FUNCTION_BLOCK "fbVFD_GSeries"   // FB120, LAD
TITLE = Controls a Siemens G120 VFD (or MicroMaster)
{ S7_Optimized_Access := 'TRUE' }
VERSION : 0.1
// stored: AutoNumber false, IsIECCheckEnabled false, IsRetainMemResEnabled false, MemoryReserve 100, SetENOAutomatically false, UDAEnableTagReadback false
   VAR_INPUT
      tInTimeout { ExternalAccessible := 'False'; ExternalVisible := 'False'; ExternalWritable := 'False'} : Time;   // Timeout Time
      iInMode { ExternalAccessible := 'False'; ExternalVisible := 'False'; ExternalWritable := 'False'} : Int;   // Mode Selection
      hwInTelegram { ExternalAccessible := 'False'; ExternalVisible := 'False'; ExternalWritable := 'False'} : HW_SUBMODULE;   // VFD Standard Telegram 1 HW address
      bInEstop { ExternalAccessible := 'False'; ExternalVisible := 'False'; ExternalWritable := 'False'} : Bool;   // Estop
      bInSignalContactor { ExternalAccessible := 'False'; ExternalVisible := 'False'; ExternalWritable := 'False'} : Bool;   // Feedback signal from Contactor
      bInEnableForward { ExternalAccessible := 'False'; ExternalVisible := 'False'; ExternalWritable := 'False'} : Bool;   // Forward motion enebled
      bInEnableReverse { ExternalAccessible := 'False'; ExternalVisible := 'False'; ExternalWritable := 'False'} : Bool := false;   // Reverse motion enabled
      rInCommandSpeed { ExternalAccessible := 'False'; ExternalVisible := 'False'; ExternalWritable := 'False'} : Real;   // Auto mode speed SP
      bInCommandForward { ExternalAccessible := 'False'; ExternalVisible := 'False'; ExternalWritable := 'False'} : Bool;   // Move forward in automatic mode
      bInCommandReverse { ExternalAccessible := 'False'; ExternalVisible := 'False'; ExternalWritable := 'False'} : Bool := false;   // Move Reverse in automatic mode
      bInResetError { ExternalAccessible := 'False'; ExternalVisible := 'False'; ExternalWritable := 'False'} : Bool;   // Reset Error
      bInMotorProtector { ExternalAccessible := 'False'; ExternalVisible := 'False'; ExternalWritable := 'False'} : Bool := true;   // Motor Protector input
      bInLocalDisconnect { ExternalAccessible := 'False'; ExternalVisible := 'False'; ExternalWritable := 'False'} : Bool := true;   // Local switch input
      bInClutch { ExternalAccessible := 'False'; ExternalVisible := 'False'; ExternalWritable := 'False'} : Bool := true;   // Overload clutch
      bInCoolingFan { ExternalAccessible := 'False'; ExternalVisible := 'False'; ExternalWritable := 'False'} : Bool := true;   // Cooling fan input
      bInUseCurrentAlarm { ExternalAccessible := 'False'; ExternalVisible := 'False'; ExternalWritable := 'False'} : Bool := false;   // True if current alarm should be active
      bInUseMaxFrequencyAlarm { ExternalAccessible := 'False'; ExternalVisible := 'False'; ExternalWritable := 'False'} : Bool := false;   // True is max frequency alarm should be active
      bInSimulate { ExternalAccessible := 'False'; ExternalVisible := 'False'; ExternalWritable := 'False'} : Bool := false;   // Activate device simulation
   END_VAR
   VAR_OUTPUT
      rOutSpeed { ExternalAccessible := 'False'; ExternalVisible := 'False'; ExternalWritable := 'False'} : Real;   // Actual motor speed
      bOutContactor { ExternalAccessible := 'False'; ExternalVisible := 'False'; ExternalWritable := 'False'} : Bool;   // Motor contactor ON
      bOutCommandForward { ExternalAccessible := 'False'; ExternalVisible := 'False'; ExternalWritable := 'False'} : Bool;   // Motor forward command
      bOutCommandReverse { ExternalAccessible := 'False'; ExternalVisible := 'False'; ExternalWritable := 'False'} : Bool := false;   // Motor reverse command
      bOutActiveForward { ExternalAccessible := 'False'; ExternalVisible := 'False'; ExternalWritable := 'False'} : Bool;   // Motor is running forward
      bOutActiveReverse { ExternalAccessible := 'False'; ExternalVisible := 'False'; ExternalWritable := 'False'} : Bool;   // Motor is running backward
      bOutAuto { ExternalAccessible := 'False'; ExternalVisible := 'False'; ExternalWritable := 'False'} : Bool;   // Block in auto mode
      bOutError { ExternalAccessible := 'False'; ExternalVisible := 'False'; ExternalWritable := 'False'} : Bool;   // Error exists
      ERROR_VFD { ExternalAccessible := 'False'; ExternalVisible := 'False'; ExternalWritable := 'False'} : "udtError_VFD";   // UDT Structure for VFD errors
   END_VAR
   VAR_IN_OUT
      HMI_VFD_Control : "udtHMI_VFD_Control";   // UDT Structure for VFD HMI control
   END_VAR
   VAR
      ErrorScroller { ExternalAccessible := 'False'; ExternalVisible := 'False'; ExternalWritable := 'False'; S7_SetPoint := 'True'} : "fbErrorScroller";   // fb to control scrolling of errors on HMI
      TON_TimeOut { ExternalAccessible := 'False'; ExternalVisible := 'False'; ExternalWritable := 'False'; S7_SetPoint := 'True'} : TON_TIME;   // Timer for Timeout time
      TON_ContactorDelay { ExternalAccessible := 'False'; ExternalVisible := 'False'; ExternalWritable := 'False'; S7_SetPoint := 'True'} : TON_TIME;   // Contactor on delay timer before check errors
      TON_CoolingFan { ExternalAccessible := 'False'; ExternalVisible := 'False'; ExternalWritable := 'False'; S7_SetPoint := 'True'} : TON_TIME;
      TON_CurrentLimitDebounce { ExternalAccessible := 'False'; ExternalVisible := 'False'; ExternalWritable := 'False'; S7_SetPoint := 'True'} : TON_TIME;   // Debounce timer for current at limit
      iLastMode { ExternalAccessible := 'False'; ExternalVisible := 'False'; ExternalWritable := 'False'} : Int;   // Last mode code
      wStatusWord { ExternalAccessible := 'False'; ExternalVisible := 'False'; ExternalWritable := 'False'} : Word;   // VFD Status word
      iActualSpeed { ExternalAccessible := 'False'; ExternalVisible := 'False'; ExternalWritable := 'False'} : Int;   // VFD Actual speed
      wControlWord { ExternalAccessible := 'False'; ExternalVisible := 'False'; ExternalWritable := 'False'} : Word;   // VFD Control word output
      iSpeedSetPoint { ExternalAccessible := 'False'; ExternalVisible := 'False'; ExternalWritable := 'False'} : Int;   // VFD Speed output
      rCommandSpeed { ExternalAccessible := 'False'; ExternalVisible := 'False'; ExternalWritable := 'False'} : Real;   // Speed command
      bNewMode { ExternalAccessible := 'False'; ExternalVisible := 'False'; ExternalWritable := 'False'} : Bool;   // New mode selected
      bEnableForward { ExternalAccessible := 'False'; ExternalVisible := 'False'; ExternalWritable := 'False'} : Bool;   // Forward enabled
      bEnableReverse { ExternalAccessible := 'False'; ExternalVisible := 'False'; ExternalWritable := 'False'} : Bool;   // Reverse enabled
      bManualMode { ExternalAccessible := 'False'; ExternalVisible := 'False'; ExternalWritable := 'False'} : Bool;   // Manual Mode is Active
      bAutoMode { ExternalAccessible := 'False'; ExternalVisible := 'False'; ExternalWritable := 'False'} : Bool;   // Auto Mode is Active
      bRunTimeoutTimer { ExternalAccessible := 'False'; ExternalVisible := 'False'; ExternalWritable := 'False'} : Bool;   // run the timeout timer
      bReset { ExternalAccessible := 'False'; ExternalVisible := 'False'; ExternalWritable := 'False'} : Bool;
      bTON_TimeOut { ExternalAccessible := 'False'; ExternalVisible := 'False'; ExternalWritable := 'False'} : Bool;
      bTON_ContactorDelay { ExternalAccessible := 'False'; ExternalVisible := 'False'; ExternalWritable := 'False'} : Bool;
      bTON_CoolingFan { ExternalAccessible := 'False'; ExternalVisible := 'False'; ExternalWritable := 'False'} : Bool;
      bTON_CurrentLimitDebounce { ExternalAccessible := 'False'; ExternalVisible := 'False'; ExternalWritable := 'False'} : Bool;
      bPB_Forward { ExternalAccessible := 'False'; ExternalVisible := 'False'; ExternalWritable := 'False'} : Bool;
      bPB_Reverse { ExternalAccessible := 'False'; ExternalVisible := 'False'; ExternalWritable := 'False'} : Bool;
      bPB_Stop { ExternalAccessible := 'False'; ExternalVisible := 'False'; ExternalWritable := 'False'} : Bool;
      bPB_ResetError { ExternalAccessible := 'False'; ExternalVisible := 'False'; ExternalWritable := 'False'} : Bool;
   END_VAR
   VAR_TEMP
      CONTROL : Struct   // VFD Control Structure
         bON : Bool;   // On
         bOFF2 : Bool;   // Off2
         bOFF3 : Bool;   // Off3
         bENABLE_OPERATION : Bool;   // Enable Operation
         bDISABLE_RFG : Bool;   // Disable RFG
         bENABLE_RFG : Bool;   // Enable RFG
         bSETPOINT_ENABLE : Bool;   // Setpoint Enable
         bFAULT_ACK : Bool;   // Fault Acknowledge
         bCW_ACTIVATION : Bool;   // CW Activation
         bCCW_ACTIVATION : Bool;   // CCW Activation
         bSP_VALID : Bool;   // SP Valid
         bSP_INVERTED : Bool;   // SP Inverted
         bSPARE01 : Bool;   // Spare
         bMOTOR_POT_UP : Bool;   // Motor Pot up
         bMOTOR_POT_DN : Bool;   // Motor Pot down
         bLOCAL_ACTIVE : Bool;   // Local Active
      END_STRUCT;
      STATUS : Struct   // VFD Status Structure
         bAT_SETPOINT_FREQ : Bool;   // At Setpoint Frequency
         bMASTER_CONTROL : Bool;   // Master Control
         bMAX_FREQ_REACHED : Bool;   // Max Frequency Reached
         bCURRENT_LIMIT : Bool;   // Current Limit
         bBRAKE_ACTIVE : Bool;   // Brake Active
         bMOTOR_OVERLOAD : Bool;   // Motor Overload
         bCW_ROTATION : Bool;   // CW Rotation
         bINVERTER_OVERLOAD : Bool;   // Inverter Overload
         bREADY_FOR_ENABLE : Bool;   // Ready for Enable
         bREADY_TO_RUN : Bool;   // Ready To Run
         bRUNNING : Bool;   // Running
         bFAULT : Bool;   // Fault
         bOFF2_ACTIVE : Bool;   // Off2 Active
         bOFF3_ACTIVE : Bool;   // Off3 Active
         bSTART_LOCKOUT : Bool;   // Start Lockout
         bALARM : Bool;   // Alarm
      END_STRUCT;
      bMajorFault : Bool;   // Major Fault
      arrReadTemp : Array[1..6] of Word;
      dwWriteTemp : DWord;   // temporary dword
      bTemp : Bool;   // temp bit
      wTempWordValue : Word;   // used for temporaily holding a word value
      iTemp : Word;
      rTemp : Real;   // temporary real value
      tTemp : Time;   // temp time value
   END_VAR
   VAR CONSTANT
      crMaxSetPoint : Real := 200.0;   // Maximum speed set point
      crMinSetPoint : Real := 0.0;   // Minimum speed set point
      crSpeedScaling : Real := 163.84;   // Reference speed scale value
   END_VAR
   VAR_TEMP   // added for the SCL form of the ladder/FBD networks
      _w1 : Bool;
      _w2 : Bool;
      _w3 : Bool;
      _w4 : Bool;
   END_VAR
BEGIN

REGION Network 1: --------------------------------------------------------- Inputs ------------------------------------------------------------------
END_REGION

REGION Network 2: Read HMI input buttons
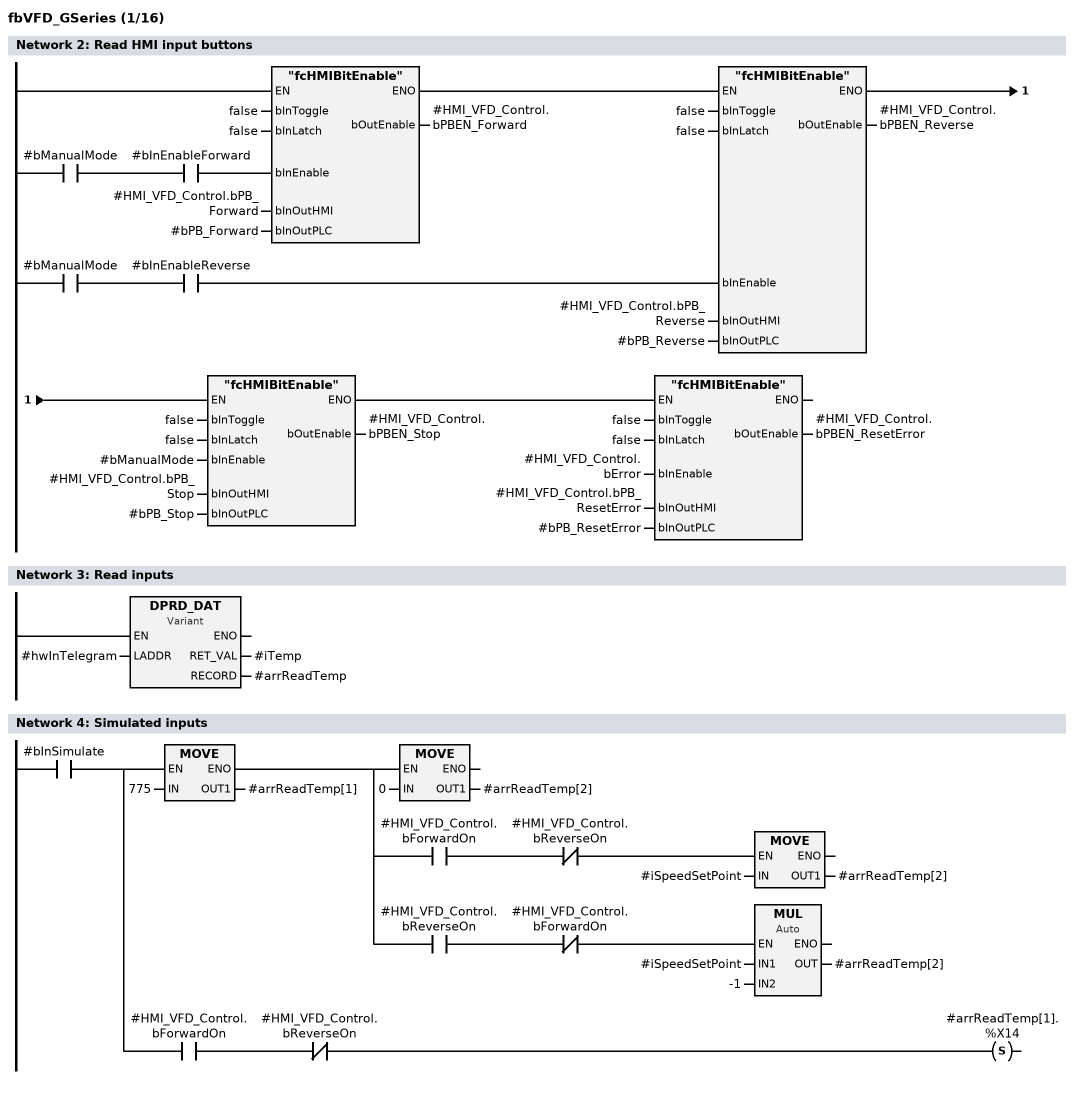
   RUNG wire#powerrail
      "fcHMIBitEnable"(bInEnable := wire#w1, bInToggle := false, bInLatch := false, bInOutHMI := #HMI_VFD_Control.bPB_Forward, bInOutPLC := #bPB_Forward, bOutEnable => #HMI_VFD_Control.bPBEN_Forward)
      "fcHMIBitEnable"(bInEnable := wire#w2, bInToggle := false, bInLatch := false, bInOutHMI := #HMI_VFD_Control.bPB_Reverse, bInOutPLC := #bPB_Reverse, bOutEnable => #HMI_VFD_Control.bPBEN_Reverse)
      "fcHMIBitEnable"(bInToggle := false, bInLatch := false, bInEnable := #bManualMode, bInOutHMI := #HMI_VFD_Control.bPB_Stop, bInOutPLC := #bPB_Stop, bOutEnable => #HMI_VFD_Control.bPBEN_Stop)
      "fcHMIBitEnable"(bInToggle := false, bInLatch := false, bInEnable := #HMI_VFD_Control.bError, bInOutHMI := #HMI_VFD_Control.bPB_ResetError, bInOutPLC := #bPB_ResetError, bOutEnable => #HMI_VFD_Control.bPBEN_ResetError)
   END_RUNG
   RUNG wire#powerrail
      Contact( #bManualMode )
      Contact( #bInEnableForward )
   END_RUNG wire#w1
   RUNG wire#powerrail
      Contact( #bManualMode )
      Contact( #bInEnableReverse )
   END_RUNG wire#w2
   // the same network as SCL:
   "fcHMIBitEnable"(bInToggle := false,
                    bInLatch := false,
                    bInEnable := #bManualMode AND #bInEnableForward,
                    bInOutHMI := #HMI_VFD_Control.bPB_Forward,
                    bInOutPLC := #bPB_Forward,
                    bOutEnable => #HMI_VFD_Control.bPBEN_Forward,
                    ENO => #_w1);
   "fcHMIBitEnable"(EN := #_w1,
                    bInToggle := false,
                    bInLatch := false,
                    bInEnable := #bManualMode AND #bInEnableReverse,
                    bInOutHMI := #HMI_VFD_Control.bPB_Reverse,
                    bInOutPLC := #bPB_Reverse,
                    bOutEnable => #HMI_VFD_Control.bPBEN_Reverse,
                    ENO => #_w2);
   "fcHMIBitEnable"(EN := #_w2,
                    bInToggle := false,
                    bInLatch := false,
                    bInEnable := #bManualMode,
                    bInOutHMI := #HMI_VFD_Control.bPB_Stop,
                    bInOutPLC := #bPB_Stop,
                    bOutEnable => #HMI_VFD_Control.bPBEN_Stop,
                    ENO => #_w3);
   IF #_w3 THEN
       "fcHMIBitEnable"(bInToggle := false,
                        bInLatch := false,
                        bInEnable := #HMI_VFD_Control.bError,
                        bInOutHMI := #HMI_VFD_Control.bPB_ResetError,
                        bInOutPLC := #bPB_ResetError,
                        bOutEnable => #HMI_VFD_Control.bPBEN_ResetError);
   END_IF;
END_REGION

REGION Network 3: Read inputs
   RUNG wire#powerrail
      { S7_Templates := "[ptr_type := Variant, laddr_type := HW_IO]" } DPRD_DAT(LADDR := #hwInTelegram, RET_VAL => #iTemp, RECORD => #arrReadTemp)
   END_RUNG
   // the same network as SCL:
   #iTemp := DPRD_DAT(LADDR := #hwInTelegram, RECORD => #arrReadTemp);
END_REGION

REGION Network 4: Simulated inputs
   RUNG wire#powerrail
      Contact( #bInSimulate )
      wire#w1
      Move(in := 775, out1 => #arrReadTemp[1])
      wire#w2
      Move(in := 0, out1 => #arrReadTemp[2])
   END_RUNG
   RUNG wire#w2
      Contact( #HMI_VFD_Control.bForwardOn )
      I_Contact( #HMI_VFD_Control.bReverseOn )
      Move(in := #iSpeedSetPoint, out1 => #arrReadTemp[2])
   END_RUNG
   RUNG wire#w2
      Contact( #HMI_VFD_Control.bReverseOn )
      I_Contact( #HMI_VFD_Control.bForwardOn )
      Mul(in1 := #iSpeedSetPoint, in2 := -1, out => #arrReadTemp[2])
   END_RUNG
   RUNG wire#w1
      Contact( #HMI_VFD_Control.bForwardOn )
      I_Contact( #HMI_VFD_Control.bReverseOn )
      S_Coil( #arrReadTemp[1].%X14 )
   END_RUNG
   // the same network as SCL:
   IF #bInSimulate THEN
       #arrReadTemp[1] := 775;
       #arrReadTemp[2] := 0;
   END_IF;
   IF #bInSimulate AND #HMI_VFD_Control.bForwardOn AND NOT #HMI_VFD_Control.bReverseOn THEN
       #arrReadTemp[2] := #iSpeedSetPoint;
   END_IF;
   IF #bInSimulate AND #HMI_VFD_Control.bReverseOn AND NOT #HMI_VFD_Control.bForwardOn THEN
       #arrReadTemp[2] := #iSpeedSetPoint * (-1);
   END_IF;
   IF #bInSimulate AND #HMI_VFD_Control.bForwardOn AND NOT #HMI_VFD_Control.bReverseOn THEN
       #arrReadTemp[1].%X14 := TRUE;
   END_IF;
END_REGION

REGION Network 5: Read the status word and parse to bits
   // // Read status word.  First word at iInAddress is the status word
   // wStatusWord := PIW[iInAddress];
   // 
   // fcWordToBits( wIN_WORD                    := wStatusWord,  // Parse status word
   //                 bOUT_BIT00                  := STATUS.bREADY_FOR_ENABLE,
   //                 bOUT_BIT01                  := STATUS.bREADY_TO_RUN,
   //                 bOUT_BIT02                  := STATUS.bRUNNING,
   //                 bOUT_BIT03                  := STATUS.bFAULT,
   //                 bOUT_BIT04                  := STATUS.bOFF2_ACTIVE,
   //                 bOUT_BIT05                  := STATUS.bOFF3_ACTIVE,
   //                 bOUT_BIT06                  := STATUS.bSTART_LOCKOUT,
   //                 bOUT_BIT07                  := STATUS.bALARM,
   //                 bOUT_BIT08                  := STATUS.bAT_SETPOINT_FREQ,
   //                 bOUT_BIT09                  := STATUS.bMASTER_CONTROL,
   //                 bOUT_BIT10                  := STATUS.bMAX_FREQ_REACHED,
   //                 bOUT_BIT11                  := STATUS.bCURRENT_LIMIT,
   //                 bOUT_BIT12                  := STATUS.bBRAKE_ACTIVE,
   //                 bOUT_BIT13                  := STATUS.bMOTOR_OVERLOAD,
   //                 bOUT_BIT14                  := STATUS.bCW_ROTATION,
   //                 bOUT_BIT15                  := STATUS.bINVERTER_OVERLOAD);
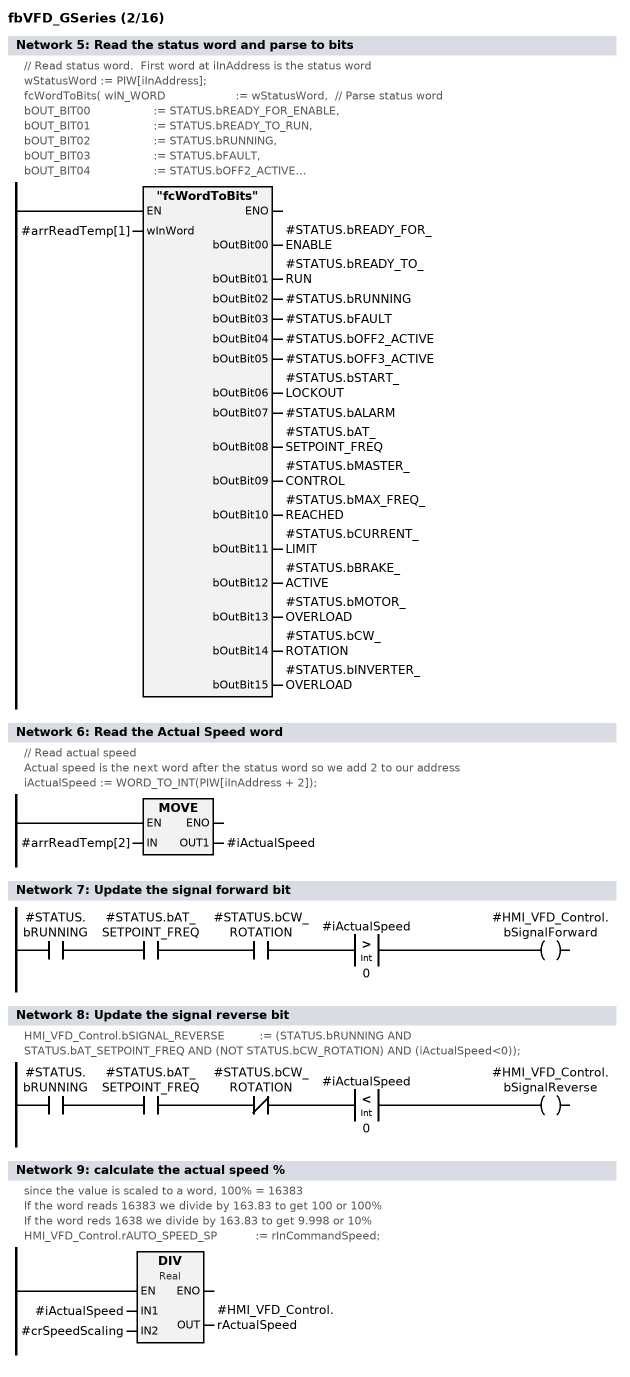
   RUNG wire#powerrail
      "fcWordToBits"(wInWord := #arrReadTemp[1], bOutBit00 => #STATUS.bREADY_FOR_ENABLE, bOutBit01 => #STATUS.bREADY_TO_RUN, bOutBit02 => #STATUS.bRUNNING, bOutBit03 => #STATUS.bFAULT, bOutBit04 => #STATUS.bOFF2_ACTIVE, bOutBit05 => #STATUS.bOFF3_ACTIVE, bOutBit06 => #STATUS.bSTART_LOCKOUT, bOutBit07 => #STATUS.bALARM, bOutBit08 => #STATUS.bAT_SETPOINT_FREQ, bOutBit09 => #STATUS.bMASTER_CONTROL, bOutBit10 => #STATUS.bMAX_FREQ_REACHED, bOutBit11 => #STATUS.bCURRENT_LIMIT, bOutBit12 => #STATUS.bBRAKE_ACTIVE, bOutBit13 => #STATUS.bMOTOR_OVERLOAD, bOutBit14 => #STATUS.bCW_ROTATION, bOutBit15 => #STATUS.bINVERTER_OVERLOAD)
   END_RUNG
   // the same network as SCL:
   "fcWordToBits"(wInWord := #arrReadTemp[1],
                  bOutBit00 => #STATUS.bREADY_FOR_ENABLE,
                  bOutBit01 => #STATUS.bREADY_TO_RUN,
                  bOutBit02 => #STATUS.bRUNNING,
                  bOutBit03 => #STATUS.bFAULT,
                  bOutBit04 => #STATUS.bOFF2_ACTIVE,
                  bOutBit05 => #STATUS.bOFF3_ACTIVE,
                  bOutBit06 => #STATUS.bSTART_LOCKOUT,
                  bOutBit07 => #STATUS.bALARM,
                  bOutBit08 => #STATUS.bAT_SETPOINT_FREQ,
                  bOutBit09 => #STATUS.bMASTER_CONTROL,
                  bOutBit10 => #STATUS.bMAX_FREQ_REACHED,
                  bOutBit11 => #STATUS.bCURRENT_LIMIT,
                  bOutBit12 => #STATUS.bBRAKE_ACTIVE,
                  bOutBit13 => #STATUS.bMOTOR_OVERLOAD,
                  bOutBit14 => #STATUS.bCW_ROTATION,
                  bOutBit15 => #STATUS.bINVERTER_OVERLOAD);
END_REGION

REGION Network 6: Read the Actual Speed word
   // // Read actual speed
   // Actual speed is the next word after the status word so we add 2 to our address
   // iActualSpeed := WORD_TO_INT(PIW[iInAddress + 2]);
   RUNG wire#powerrail
      Move(in := #arrReadTemp[2], out1 => #iActualSpeed)
   END_RUNG
   // the same network as SCL:
   #iActualSpeed := #arrReadTemp[2];
END_REGION

REGION Network 7: Update the signal forward bit
   RUNG wire#powerrail
      Contact( #STATUS.bRUNNING )
      Contact( #STATUS.bAT_SETPOINT_FREQ )
      Contact( #STATUS.bCW_ROTATION )
      { S7_Templates := "SrcType := Int" } GT_Contact(in1 := #iActualSpeed, in2 := 0)
      Coil( #HMI_VFD_Control.bSignalForward )
   END_RUNG
   // the same network as SCL:
   #HMI_VFD_Control.bSignalForward := #STATUS.bRUNNING AND #STATUS.bAT_SETPOINT_FREQ AND #STATUS.bCW_ROTATION AND (#iActualSpeed > 0);
END_REGION

REGION Network 8: Update the signal reverse bit
   // HMI_VFD_Control.bSIGNAL_REVERSE          := (STATUS.bRUNNING AND 
   // STATUS.bAT_SETPOINT_FREQ AND (NOT STATUS.bCW_ROTATION) AND (iActualSpeed<0));
   RUNG wire#powerrail
      Contact( #STATUS.bRUNNING )
      Contact( #STATUS.bAT_SETPOINT_FREQ )
      I_Contact( #STATUS.bCW_ROTATION )
      { S7_Templates := "SrcType := Int" } LT_Contact(in1 := #iActualSpeed, in2 := 0)
      Coil( #HMI_VFD_Control.bSignalReverse )
   END_RUNG
   // the same network as SCL:
   #HMI_VFD_Control.bSignalReverse := #STATUS.bRUNNING AND #STATUS.bAT_SETPOINT_FREQ AND NOT #STATUS.bCW_ROTATION AND (#iActualSpeed < 0);
END_REGION

REGION Network 9: calculate the actual speed %
   // since the value is scaled to a word, 100% = 16383
   // 
   // If the word reads 16383 we divide by 163.83 to get 100 or 100%
   // If the word reds 1638 we divide by 163.83 to get 9.998 or 10%
   // 
   // HMI_VFD_Control.rAUTO_SPEED_SP           := rInCommandSpeed;
   RUNG wire#powerrail
      { S7_Templates := "SrcType := Real" } Div(in1 := #iActualSpeed, in2 := #crSpeedScaling, out => #HMI_VFD_Control.rActualSpeed)
   END_RUNG
   // the same network as SCL:
   #HMI_VFD_Control.rActualSpeed := #iActualSpeed / #crSpeedScaling;
END_REGION

REGION Network 10: Set the automatic mode speed set point
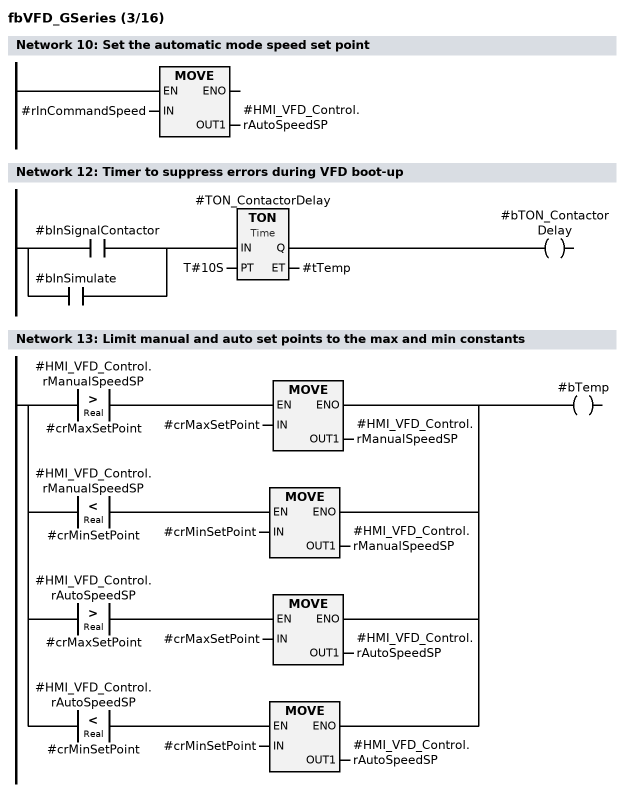
   RUNG wire#powerrail
      Move(in := #rInCommandSpeed, out1 => #HMI_VFD_Control.rAutoSpeedSP)
   END_RUNG
   // the same network as SCL:
   #HMI_VFD_Control.rAutoSpeedSP := #rInCommandSpeed;
END_REGION

REGION Network 11: --------------------------------------------------- Control Logic ------------------------------------------------------------
END_REGION

REGION Network 12: Timer to suppress errors during VFD boot-up
   RUNG wire#powerrail
      Contact( #bInSignalContactor )
      wire#w1
      { S7_Templates := "time_type := Time" } #TON_ContactorDelay.TON(pt := T#10S, et => #tTemp)
      Coil( #bTON_ContactorDelay )
   END_RUNG
   RUNG wire#powerrail
      Contact( #bInSimulate )
   END_RUNG wire#w1
   // the same network as SCL:
   #TON_ContactorDelay(IN := #bInSignalContactor OR #bInSimulate, PT := T#10S, ET => #tTemp);   // TON
   #bTON_ContactorDelay := #TON_ContactorDelay.Q;
END_REGION

REGION Network 13: Limit manual and auto set points to the max and min constants
   RUNG wire#powerrail
      { S7_Templates := "SrcType := Real" } GT_Contact(in1 := #HMI_VFD_Control.rManualSpeedSP, in2 := #crMaxSetPoint)
      Move(in := #crMaxSetPoint, out1 => #HMI_VFD_Control.rManualSpeedSP)
      wire#w1
      Coil( #bTemp )
   END_RUNG
   RUNG wire#powerrail
      { S7_Templates := "SrcType := Real" } LT_Contact(in1 := #HMI_VFD_Control.rManualSpeedSP, in2 := #crMinSetPoint)
      Move(in := #crMinSetPoint, out1 => #HMI_VFD_Control.rManualSpeedSP)
   END_RUNG wire#w1
   RUNG wire#powerrail
      { S7_Templates := "SrcType := Real" } GT_Contact(in1 := #HMI_VFD_Control.rAutoSpeedSP, in2 := #crMaxSetPoint)
      Move(in := #crMaxSetPoint, out1 => #HMI_VFD_Control.rAutoSpeedSP)
   END_RUNG wire#w1
   RUNG wire#powerrail
      { S7_Templates := "SrcType := Real" } LT_Contact(in1 := #HMI_VFD_Control.rAutoSpeedSP, in2 := #crMinSetPoint)
      Move(in := #crMinSetPoint, out1 => #HMI_VFD_Control.rAutoSpeedSP)
   END_RUNG wire#w1
   // the same network as SCL:
   #_w1 := #HMI_VFD_Control.rManualSpeedSP > #crMaxSetPoint;
   IF #_w1 THEN #HMI_VFD_Control.rManualSpeedSP := #crMaxSetPoint; END_IF;
   #_w2 := #HMI_VFD_Control.rManualSpeedSP < #crMinSetPoint;
   IF #_w2 THEN #HMI_VFD_Control.rManualSpeedSP := #crMinSetPoint; END_IF;
   #_w3 := #HMI_VFD_Control.rAutoSpeedSP > #crMaxSetPoint;
   IF #_w3 THEN #HMI_VFD_Control.rAutoSpeedSP := #crMaxSetPoint; END_IF;
   #_w4 := #HMI_VFD_Control.rAutoSpeedSP < #crMinSetPoint;
   IF #_w4 THEN #HMI_VFD_Control.rAutoSpeedSP := #crMinSetPoint; END_IF;
   #bTemp := #_w1 OR #_w2 OR #_w3 OR #_w4;
END_REGION

REGION Network 14: Reset errors
   // Clear all errors
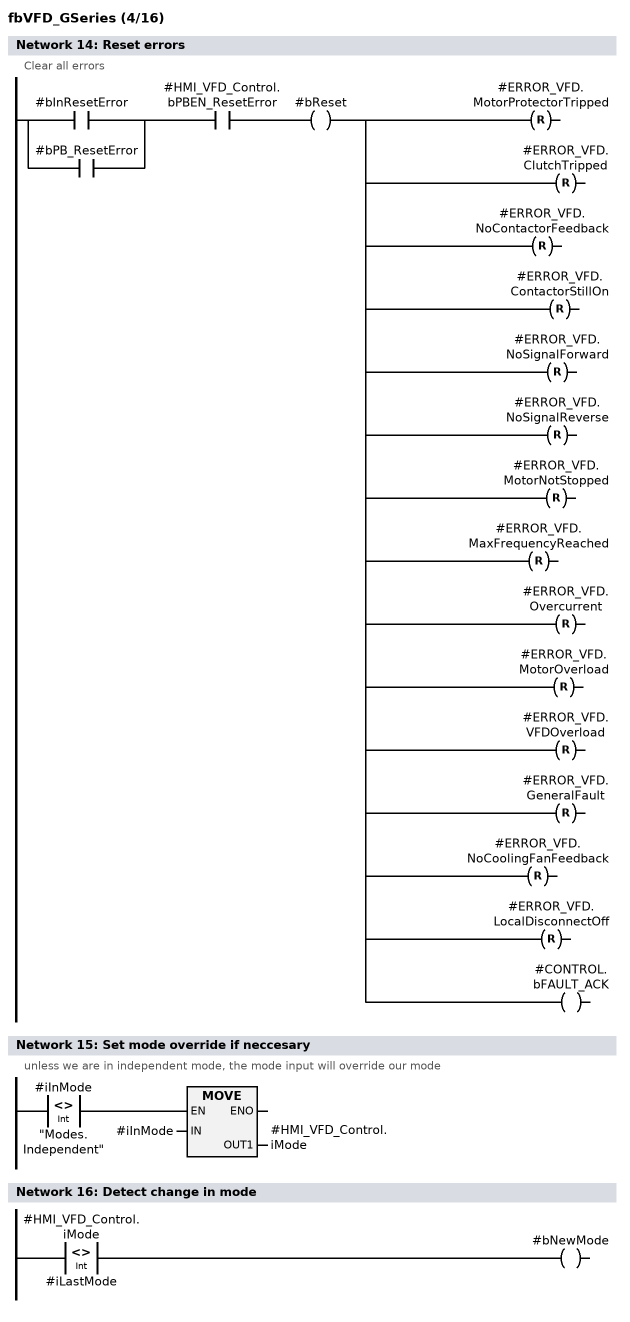
   RUNG wire#powerrail
      Contact( #bInResetError )
      wire#w1
      Contact( #HMI_VFD_Control.bPBEN_ResetError )
      Coil( #bReset )
      wire#w2
      R_Coil( #ERROR_VFD.MotorProtectorTripped )
   END_RUNG
   RUNG wire#powerrail
      Contact( #bPB_ResetError )
   END_RUNG wire#w1
   RUNG wire#w2
      R_Coil( #ERROR_VFD.ClutchTripped )
   END_RUNG
   RUNG wire#w2
      R_Coil( #ERROR_VFD.NoContactorFeedback )
   END_RUNG
   RUNG wire#w2
      R_Coil( #ERROR_VFD.ContactorStillOn )
   END_RUNG
   RUNG wire#w2
      R_Coil( #ERROR_VFD.NoSignalForward )
   END_RUNG
   RUNG wire#w2
      R_Coil( #ERROR_VFD.NoSignalReverse )
   END_RUNG
   RUNG wire#w2
      R_Coil( #ERROR_VFD.MotorNotStopped )
   END_RUNG
   RUNG wire#w2
      R_Coil( #ERROR_VFD.MaxFrequencyReached )
   END_RUNG
   RUNG wire#w2
      R_Coil( #ERROR_VFD.Overcurrent )
   END_RUNG
   RUNG wire#w2
      R_Coil( #ERROR_VFD.MotorOverload )
   END_RUNG
   RUNG wire#w2
      R_Coil( #ERROR_VFD.VFDOverload )
   END_RUNG
   RUNG wire#w2
      R_Coil( #ERROR_VFD.GeneralFault )
   END_RUNG
   RUNG wire#w2
      R_Coil( #ERROR_VFD.NoCoolingFanFeedback )
   END_RUNG
   RUNG wire#w2
      R_Coil( #ERROR_VFD.LocalDisconnectOff )
   END_RUNG
   RUNG wire#w2
      Coil( #CONTROL.bFAULT_ACK )
   END_RUNG
   // the same network as SCL:
   #bReset := (#bInResetError OR #bPB_ResetError) AND #HMI_VFD_Control.bPBEN_ResetError;
   IF #bReset THEN
       #ERROR_VFD.MotorProtectorTripped := FALSE;
       #ERROR_VFD.ClutchTripped := FALSE;
       #ERROR_VFD.NoContactorFeedback := FALSE;
       #ERROR_VFD.ContactorStillOn := FALSE;
       #ERROR_VFD.NoSignalForward := FALSE;
       #ERROR_VFD.NoSignalReverse := FALSE;
       #ERROR_VFD.MotorNotStopped := FALSE;
       #ERROR_VFD.MaxFrequencyReached := FALSE;
       #ERROR_VFD.Overcurrent := FALSE;
       #ERROR_VFD.MotorOverload := FALSE;
       #ERROR_VFD.VFDOverload := FALSE;
       #ERROR_VFD.GeneralFault := FALSE;
       #ERROR_VFD.NoCoolingFanFeedback := FALSE;
       #ERROR_VFD.LocalDisconnectOff := FALSE;
   END_IF;
   #CONTROL.bFAULT_ACK := #bReset;
END_REGION

REGION Network 15: Set mode override if neccesary
   // unless we are in independent mode, the mode input will override our mode
   RUNG wire#powerrail
      { S7_Templates := "SrcType := Int" } NE_Contact(in1 := #iInMode, in2 := "Modes.Independent")
      Move(in := #iInMode, out1 => #HMI_VFD_Control.iMode)
   END_RUNG
   // the same network as SCL:
   IF #iInMode <> "Modes.Independent" THEN #HMI_VFD_Control.iMode := #iInMode; END_IF;
END_REGION

REGION Network 16: Detect change in mode
   RUNG wire#powerrail
      { S7_Templates := "SrcType := Int" } NE_Contact(in1 := #HMI_VFD_Control.iMode, in2 := #iLastMode)
      Coil( #bNewMode )
   END_RUNG
   // the same network as SCL:
   #bNewMode := #HMI_VFD_Control.iMode <> #iLastMode;
END_REGION

REGION Network 17: Keep track of last mode
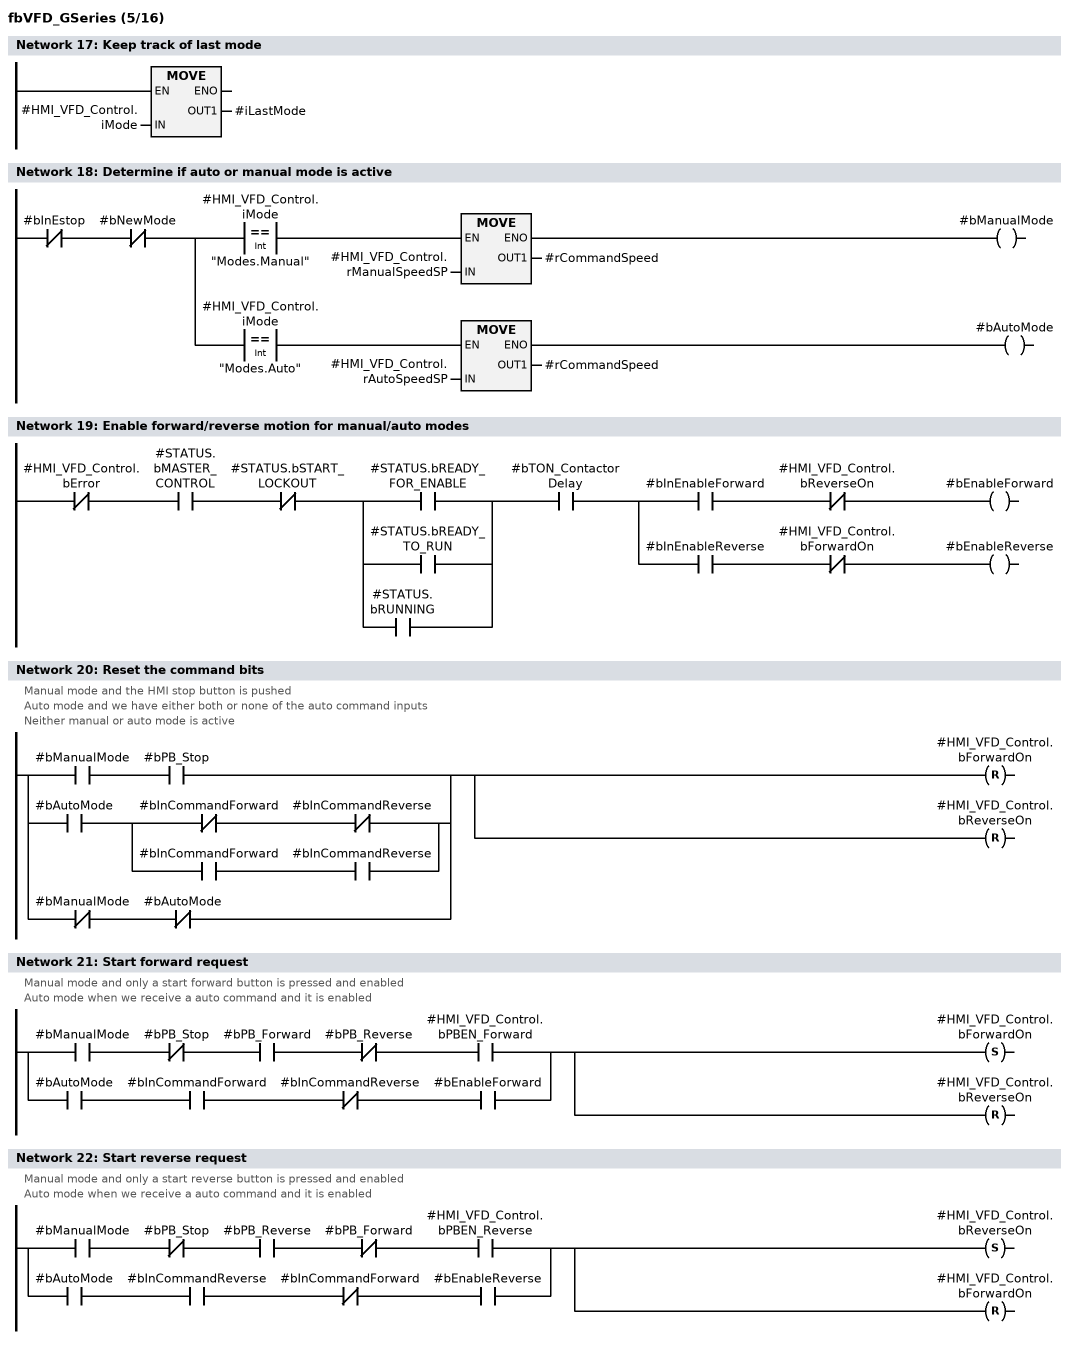
   RUNG wire#powerrail
      Move(in := #HMI_VFD_Control.iMode, out1 => #iLastMode)
   END_RUNG
   // the same network as SCL:
   #iLastMode := #HMI_VFD_Control.iMode;
END_REGION

REGION Network 18: Determine if auto or manual mode is active
   RUNG wire#powerrail
      I_Contact( #bInEstop )
      I_Contact( #bNewMode )
      wire#w1
      { S7_Templates := "SrcType := Int" } EQ_Contact(in1 := #HMI_VFD_Control.iMode, in2 := "Modes.Manual")
      Move(in := #HMI_VFD_Control.rManualSpeedSP, out1 => #rCommandSpeed)
      Coil( #bManualMode )
   END_RUNG
   RUNG wire#w1
      { S7_Templates := "SrcType := Int" } EQ_Contact(in1 := #HMI_VFD_Control.iMode, in2 := "Modes.Auto")
      Move(in := #HMI_VFD_Control.rAutoSpeedSP, out1 => #rCommandSpeed)
      Coil( #bAutoMode )
   END_RUNG
   // the same network as SCL:
   #_w1 := NOT #bInEstop AND NOT #bNewMode;
   #_w2 := #_w1 AND (#HMI_VFD_Control.iMode = "Modes.Manual");
   IF #_w2 THEN #rCommandSpeed := #HMI_VFD_Control.rManualSpeedSP; END_IF;
   #bManualMode := #_w2;
   #_w3 := #_w1 AND (#HMI_VFD_Control.iMode = "Modes.Auto");
   IF #_w3 THEN #rCommandSpeed := #HMI_VFD_Control.rAutoSpeedSP; END_IF;
   #bAutoMode := #_w3;
END_REGION

REGION Network 19: Enable forward/reverse motion for manual/auto modes
   RUNG wire#powerrail
      I_Contact( #HMI_VFD_Control.bError )
      Contact( #STATUS.bMASTER_CONTROL )
      I_Contact( #STATUS.bSTART_LOCKOUT )
      wire#w1
      Contact( #STATUS.bREADY_FOR_ENABLE )
      wire#w2
      Contact( #bTON_ContactorDelay )
      wire#w3
      Contact( #bInEnableForward )
      I_Contact( #HMI_VFD_Control.bReverseOn )
      Coil( #bEnableForward )
   END_RUNG
   RUNG wire#w1
      Contact( #STATUS.bREADY_TO_RUN )
   END_RUNG wire#w2
   RUNG wire#w1
      Contact( #STATUS.bRUNNING )
   END_RUNG wire#w2
   RUNG wire#w3
      Contact( #bInEnableReverse )
      I_Contact( #HMI_VFD_Control.bForwardOn )
      Coil( #bEnableReverse )
   END_RUNG
   // the same network as SCL:
   #_w1 := NOT #HMI_VFD_Control.bError AND #STATUS.bMASTER_CONTROL AND NOT #STATUS.bSTART_LOCKOUT AND (#STATUS.bREADY_FOR_ENABLE OR #STATUS.bREADY_TO_RUN OR #STATUS.bRUNNING) AND #bTON_ContactorDelay;
   #bEnableForward := #_w1 AND #bInEnableForward AND NOT #HMI_VFD_Control.bReverseOn;
   #bEnableReverse := #_w1 AND #bInEnableReverse AND NOT #HMI_VFD_Control.bForwardOn;
END_REGION

REGION Network 20: Reset the command bits
   // Manual mode and the HMI stop button is pushed
   // Auto mode and we have either both or none of the auto command inputs
   // Neither manual or auto mode is active
   RUNG wire#powerrail
      Contact( #bManualMode )
      Contact( #bPB_Stop )
      wire#w1
      R_Coil( #HMI_VFD_Control.bForwardOn )
   END_RUNG
   RUNG wire#powerrail
      Contact( #bAutoMode )
      wire#w2
      I_Contact( #bInCommandForward )
      I_Contact( #bInCommandReverse )
   END_RUNG wire#w1
   RUNG wire#w2
      Contact( #bInCommandForward )
      Contact( #bInCommandReverse )
   END_RUNG wire#w1
   RUNG wire#powerrail
      I_Contact( #bManualMode )
      I_Contact( #bAutoMode )
   END_RUNG wire#w1
   RUNG wire#w1
      R_Coil( #HMI_VFD_Control.bReverseOn )
   END_RUNG
   // the same network as SCL:
   IF (#bManualMode AND #bPB_Stop) OR (#bAutoMode AND ((NOT #bInCommandForward AND NOT #bInCommandReverse) OR (#bInCommandForward AND #bInCommandReverse))) OR (NOT #bManualMode AND NOT #bAutoMode) THEN
       #HMI_VFD_Control.bForwardOn := FALSE;
       #HMI_VFD_Control.bReverseOn := FALSE;
   END_IF;
END_REGION

REGION Network 21: Start forward request
   // Manual mode and only a start forward button is pressed and enabled
   // Auto mode when we receive a auto command and it is enabled
   RUNG wire#powerrail
      Contact( #bManualMode )
      I_Contact( #bPB_Stop )
      Contact( #bPB_Forward )
      I_Contact( #bPB_Reverse )
      Contact( #HMI_VFD_Control.bPBEN_Forward )
      wire#w1
      S_Coil( #HMI_VFD_Control.bForwardOn )
   END_RUNG
   RUNG wire#powerrail
      Contact( #bAutoMode )
      Contact( #bInCommandForward )
      I_Contact( #bInCommandReverse )
      Contact( #bEnableForward )
   END_RUNG wire#w1
   RUNG wire#w1
      R_Coil( #HMI_VFD_Control.bReverseOn )
   END_RUNG
   // the same network as SCL:
   IF (#bManualMode AND NOT #bPB_Stop AND #bPB_Forward AND NOT #bPB_Reverse AND #HMI_VFD_Control.bPBEN_Forward) OR (#bAutoMode AND #bInCommandForward AND NOT #bInCommandReverse AND #bEnableForward) THEN
       #HMI_VFD_Control.bForwardOn := TRUE;
       #HMI_VFD_Control.bReverseOn := FALSE;
   END_IF;
END_REGION

REGION Network 22: Start reverse request
   // Manual mode and only a start reverse button is pressed and enabled
   // Auto mode when we receive a auto command and it is enabled
   RUNG wire#powerrail
      Contact( #bManualMode )
      I_Contact( #bPB_Stop )
      Contact( #bPB_Reverse )
      I_Contact( #bPB_Forward )
      Contact( #HMI_VFD_Control.bPBEN_Reverse )
      wire#w1
      S_Coil( #HMI_VFD_Control.bReverseOn )
   END_RUNG
   RUNG wire#powerrail
      Contact( #bAutoMode )
      Contact( #bInCommandReverse )
      I_Contact( #bInCommandForward )
      Contact( #bEnableReverse )
   END_RUNG wire#w1
   RUNG wire#w1
      R_Coil( #HMI_VFD_Control.bForwardOn )
   END_RUNG
   // the same network as SCL:
   IF (#bManualMode AND NOT #bPB_Stop AND #bPB_Reverse AND NOT #bPB_Forward AND #HMI_VFD_Control.bPBEN_Reverse) OR (#bAutoMode AND #bInCommandReverse AND NOT #bInCommandForward AND #bEnableReverse) THEN
       #HMI_VFD_Control.bReverseOn := TRUE;
       #HMI_VFD_Control.bForwardOn := FALSE;
   END_IF;
END_REGION

REGION Network 23: If the forward enable is lost, stop the forward motion
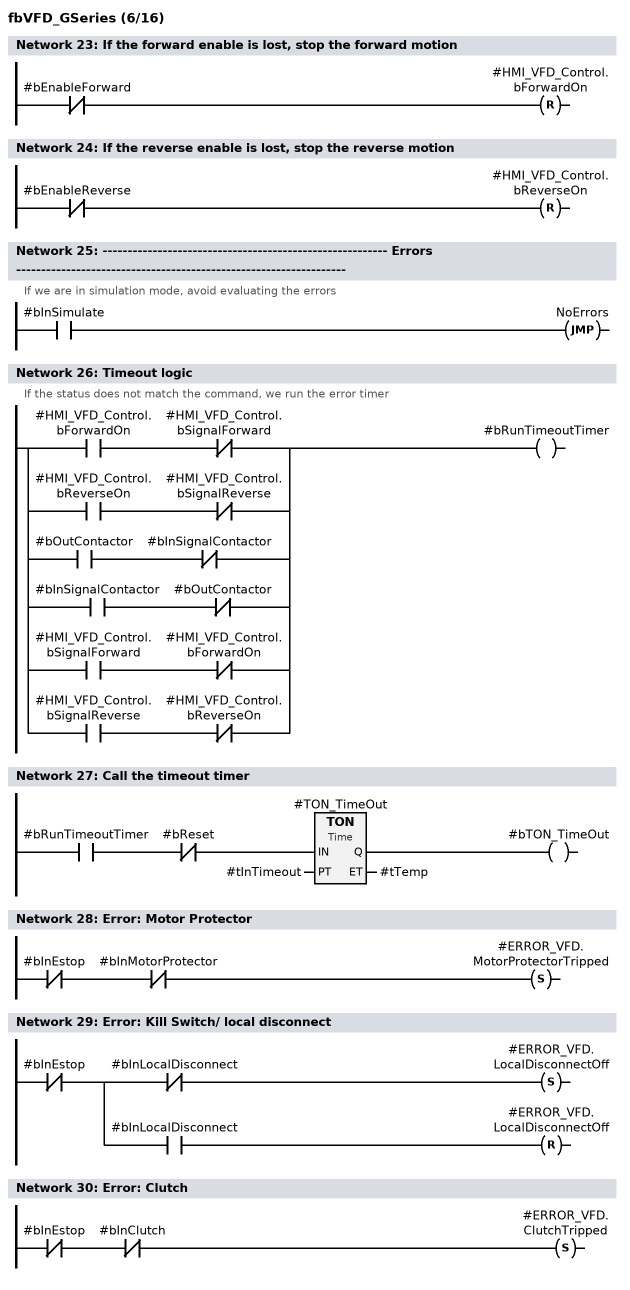
   RUNG wire#powerrail
      I_Contact( #bEnableForward )
      R_Coil( #HMI_VFD_Control.bForwardOn )
   END_RUNG
   // the same network as SCL:
   IF NOT #bEnableForward THEN #HMI_VFD_Control.bForwardOn := FALSE; END_IF;
END_REGION

REGION Network 24: If the reverse enable is lost, stop the reverse motion
   RUNG wire#powerrail
      I_Contact( #bEnableReverse )
      R_Coil( #HMI_VFD_Control.bReverseOn )
   END_RUNG
   // the same network as SCL:
   IF NOT #bEnableReverse THEN #HMI_VFD_Control.bReverseOn := FALSE; END_IF;
END_REGION

REGION Network 25: --------------------------------------------------------- Errors ------------------------------------------------------------------
   // If we are in simulation mode, avoid evaluating the errors
   RUNG wire#powerrail
      Contact( #bInSimulate )
      JumpCoil( NoErrors )
   END_RUNG
   // the same network as SCL:
   IF #bInSimulate THEN GOTO NoErrors; END_IF;
END_REGION

REGION Network 26: Timeout logic
   // If the status does not match the command, we run the error timer
   RUNG wire#powerrail
      Contact( #HMI_VFD_Control.bForwardOn )
      I_Contact( #HMI_VFD_Control.bSignalForward )
      wire#w1
      Coil( #bRunTimeoutTimer )
   END_RUNG
   RUNG wire#powerrail
      Contact( #HMI_VFD_Control.bReverseOn )
      I_Contact( #HMI_VFD_Control.bSignalReverse )
   END_RUNG wire#w1
   RUNG wire#powerrail
      Contact( #bOutContactor )
      I_Contact( #bInSignalContactor )
   END_RUNG wire#w1
   RUNG wire#powerrail
      Contact( #bInSignalContactor )
      I_Contact( #bOutContactor )
   END_RUNG wire#w1
   RUNG wire#powerrail
      Contact( #HMI_VFD_Control.bSignalForward )
      I_Contact( #HMI_VFD_Control.bForwardOn )
   END_RUNG wire#w1
   RUNG wire#powerrail
      Contact( #HMI_VFD_Control.bSignalReverse )
      I_Contact( #HMI_VFD_Control.bReverseOn )
   END_RUNG wire#w1
   // the same network as SCL:
   #bRunTimeoutTimer := (#HMI_VFD_Control.bForwardOn AND NOT #HMI_VFD_Control.bSignalForward) OR (#HMI_VFD_Control.bReverseOn AND NOT #HMI_VFD_Control.bSignalReverse) OR (#bOutContactor AND NOT #bInSignalContactor) OR (#bInSignalContactor AND NOT #bOutContactor) OR (#HMI_VFD_Control.bSignalForward AND NOT #HMI_VFD_Control.bForwardOn) OR (#HMI_VFD_Control.bSignalReverse AND NOT #HMI_VFD_Control.bReverseOn);
END_REGION

REGION Network 27: Call the timeout timer
   RUNG wire#powerrail
      Contact( #bRunTimeoutTimer )
      I_Contact( #bReset )
      { S7_Templates := "time_type := Time" } #TON_TimeOut.TON(pt := #tInTimeout, et => #tTemp)
      Coil( #bTON_TimeOut )
   END_RUNG
   // the same network as SCL:
   #TON_TimeOut(IN := #bRunTimeoutTimer AND NOT #bReset, PT := #tInTimeout, ET => #tTemp);   // TON
   #bTON_TimeOut := #TON_TimeOut.Q;
END_REGION

REGION Network 28: Error: Motor Protector
   RUNG wire#powerrail
      I_Contact( #bInEstop )
      I_Contact( #bInMotorProtector )
      S_Coil( #ERROR_VFD.MotorProtectorTripped )
   END_RUNG
   // the same network as SCL:
   IF NOT #bInEstop AND NOT #bInMotorProtector THEN #ERROR_VFD.MotorProtectorTripped := TRUE; END_IF;
END_REGION

REGION Network 29: Error: Kill Switch/ local disconnect
   RUNG wire#powerrail
      I_Contact( #bInEstop )
      wire#w1
      I_Contact( #bInLocalDisconnect )
      S_Coil( #ERROR_VFD.LocalDisconnectOff )
   END_RUNG
   RUNG wire#w1
      Contact( #bInLocalDisconnect )
      R_Coil( #ERROR_VFD.LocalDisconnectOff )
   END_RUNG
   // the same network as SCL:
   IF NOT #bInEstop AND NOT #bInLocalDisconnect THEN #ERROR_VFD.LocalDisconnectOff := TRUE; END_IF;
   IF NOT #bInEstop AND #bInLocalDisconnect THEN #ERROR_VFD.LocalDisconnectOff := FALSE; END_IF;
END_REGION

REGION Network 30: Error: Clutch
   RUNG wire#powerrail
      I_Contact( #bInEstop )
      I_Contact( #bInClutch )
      S_Coil( #ERROR_VFD.ClutchTripped )
   END_RUNG
   // the same network as SCL:
   IF NOT #bInEstop AND NOT #bInClutch THEN #ERROR_VFD.ClutchTripped := TRUE; END_IF;
END_REGION

REGION Network 31: Error: Max Frequency. This error isn't always used.
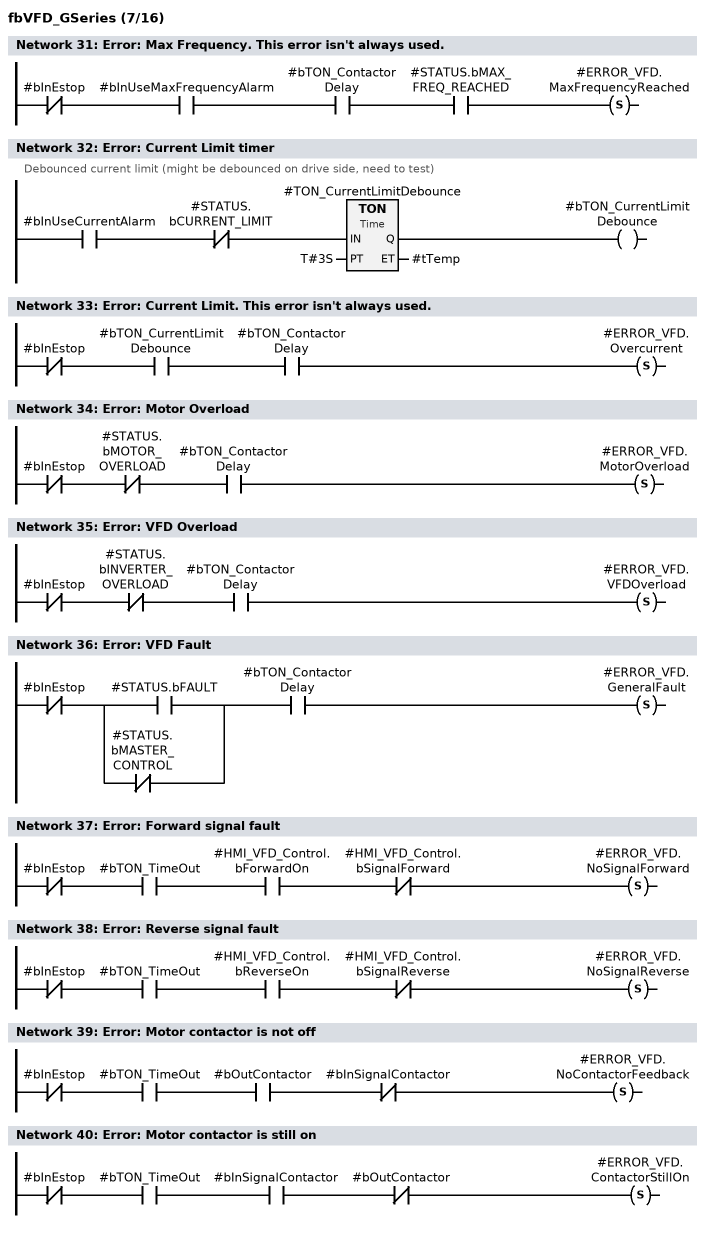
   RUNG wire#powerrail
      I_Contact( #bInEstop )
      Contact( #bInUseMaxFrequencyAlarm )
      Contact( #bTON_ContactorDelay )
      Contact( #STATUS.bMAX_FREQ_REACHED )
      S_Coil( #ERROR_VFD.MaxFrequencyReached )
   END_RUNG
   // the same network as SCL:
   IF NOT #bInEstop AND #bInUseMaxFrequencyAlarm AND #bTON_ContactorDelay AND #STATUS.bMAX_FREQ_REACHED THEN
       #ERROR_VFD.MaxFrequencyReached := TRUE;
   END_IF;
END_REGION

REGION Network 32: Error: Current Limit timer
   // Debounced current limit (might be debounced on drive side, need to test)
   RUNG wire#powerrail
      Contact( #bInUseCurrentAlarm )
      I_Contact( #STATUS.bCURRENT_LIMIT )
      { S7_Templates := "time_type := Time" } #TON_CurrentLimitDebounce.TON(pt := T#3S, et => #tTemp)
      Coil( #bTON_CurrentLimitDebounce )
   END_RUNG
   // the same network as SCL:
   #TON_CurrentLimitDebounce(IN := #bInUseCurrentAlarm AND NOT #STATUS.bCURRENT_LIMIT, PT := T#3S, ET => #tTemp);   // TON
   #bTON_CurrentLimitDebounce := #TON_CurrentLimitDebounce.Q;
END_REGION

REGION Network 33: Error: Current Limit. This error isn't always used.
   RUNG wire#powerrail
      I_Contact( #bInEstop )
      Contact( #bTON_CurrentLimitDebounce )
      Contact( #bTON_ContactorDelay )
      S_Coil( #ERROR_VFD.Overcurrent )
   END_RUNG
   // the same network as SCL:
   IF NOT #bInEstop AND #bTON_CurrentLimitDebounce AND #bTON_ContactorDelay THEN
       #ERROR_VFD.Overcurrent := TRUE;
   END_IF;
END_REGION

REGION Network 34: Error: Motor Overload
   RUNG wire#powerrail
      I_Contact( #bInEstop )
      I_Contact( #STATUS.bMOTOR_OVERLOAD )
      Contact( #bTON_ContactorDelay )
      S_Coil( #ERROR_VFD.MotorOverload )
   END_RUNG
   // the same network as SCL:
   IF NOT #bInEstop AND NOT #STATUS.bMOTOR_OVERLOAD AND #bTON_ContactorDelay THEN
       #ERROR_VFD.MotorOverload := TRUE;
   END_IF;
END_REGION

REGION Network 35: Error: VFD Overload
   RUNG wire#powerrail
      I_Contact( #bInEstop )
      I_Contact( #STATUS.bINVERTER_OVERLOAD )
      Contact( #bTON_ContactorDelay )
      S_Coil( #ERROR_VFD.VFDOverload )
   END_RUNG
   // the same network as SCL:
   IF NOT #bInEstop AND NOT #STATUS.bINVERTER_OVERLOAD AND #bTON_ContactorDelay THEN
       #ERROR_VFD.VFDOverload := TRUE;
   END_IF;
END_REGION

REGION Network 36: Error: VFD Fault
   RUNG wire#powerrail
      I_Contact( #bInEstop )
      wire#w1
      Contact( #STATUS.bFAULT )
      wire#w2
      Contact( #bTON_ContactorDelay )
      S_Coil( #ERROR_VFD.GeneralFault )
   END_RUNG
   RUNG wire#w1
      I_Contact( #STATUS.bMASTER_CONTROL )
   END_RUNG wire#w2
   // the same network as SCL:
   IF NOT #bInEstop AND (#STATUS.bFAULT OR NOT #STATUS.bMASTER_CONTROL) AND #bTON_ContactorDelay THEN
       #ERROR_VFD.GeneralFault := TRUE;
   END_IF;
END_REGION

REGION Network 37: Error: Forward signal fault
   RUNG wire#powerrail
      I_Contact( #bInEstop )
      Contact( #bTON_TimeOut )
      Contact( #HMI_VFD_Control.bForwardOn )
      I_Contact( #HMI_VFD_Control.bSignalForward )
      S_Coil( #ERROR_VFD.NoSignalForward )
   END_RUNG
   // the same network as SCL:
   IF NOT #bInEstop AND #bTON_TimeOut AND #HMI_VFD_Control.bForwardOn AND NOT #HMI_VFD_Control.bSignalForward THEN
       #ERROR_VFD.NoSignalForward := TRUE;
   END_IF;
END_REGION

REGION Network 38: Error: Reverse signal fault
   RUNG wire#powerrail
      I_Contact( #bInEstop )
      Contact( #bTON_TimeOut )
      Contact( #HMI_VFD_Control.bReverseOn )
      I_Contact( #HMI_VFD_Control.bSignalReverse )
      S_Coil( #ERROR_VFD.NoSignalReverse )
   END_RUNG
   // the same network as SCL:
   IF NOT #bInEstop AND #bTON_TimeOut AND #HMI_VFD_Control.bReverseOn AND NOT #HMI_VFD_Control.bSignalReverse THEN
       #ERROR_VFD.NoSignalReverse := TRUE;
   END_IF;
END_REGION

REGION Network 39: Error: Motor contactor is not off
   RUNG wire#powerrail
      I_Contact( #bInEstop )
      Contact( #bTON_TimeOut )
      Contact( #bOutContactor )
      I_Contact( #bInSignalContactor )
      S_Coil( #ERROR_VFD.NoContactorFeedback )
   END_RUNG
   // the same network as SCL:
   IF NOT #bInEstop AND #bTON_TimeOut AND #bOutContactor AND NOT #bInSignalContactor THEN
       #ERROR_VFD.NoContactorFeedback := TRUE;
   END_IF;
END_REGION

REGION Network 40: Error: Motor contactor is still on
   RUNG wire#powerrail
      I_Contact( #bInEstop )
      Contact( #bTON_TimeOut )
      Contact( #bInSignalContactor )
      I_Contact( #bOutContactor )
      S_Coil( #ERROR_VFD.ContactorStillOn )
   END_RUNG
   // the same network as SCL:
   IF NOT #bInEstop AND #bTON_TimeOut AND #bInSignalContactor AND NOT #bOutContactor THEN
       #ERROR_VFD.ContactorStillOn := TRUE;
   END_IF;
END_REGION

REGION Network 41: Error: Motor Doesn't stop
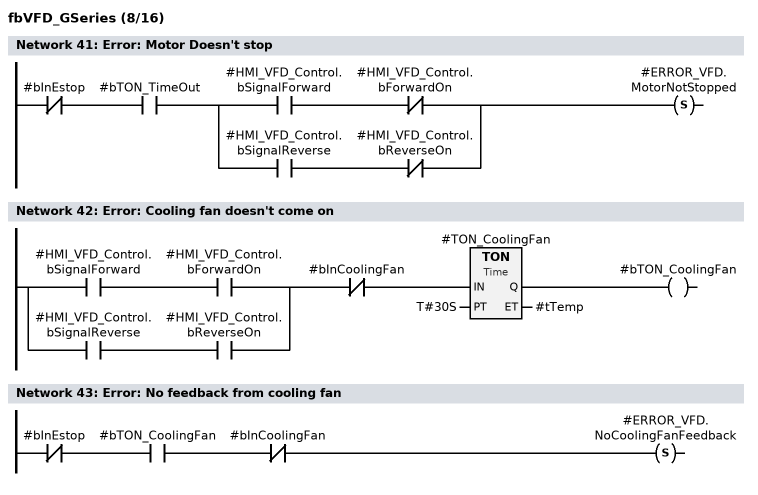
   RUNG wire#powerrail
      I_Contact( #bInEstop )
      Contact( #bTON_TimeOut )
      wire#w1
      Contact( #HMI_VFD_Control.bSignalForward )
      I_Contact( #HMI_VFD_Control.bForwardOn )
      wire#w2
      S_Coil( #ERROR_VFD.MotorNotStopped )
   END_RUNG
   RUNG wire#w1
      Contact( #HMI_VFD_Control.bSignalReverse )
      I_Contact( #HMI_VFD_Control.bReverseOn )
   END_RUNG wire#w2
   // the same network as SCL:
   IF NOT #bInEstop AND #bTON_TimeOut AND ((#HMI_VFD_Control.bSignalForward AND NOT #HMI_VFD_Control.bForwardOn) OR (#HMI_VFD_Control.bSignalReverse AND NOT #HMI_VFD_Control.bReverseOn)) THEN
       #ERROR_VFD.MotorNotStopped := TRUE;
   END_IF;
END_REGION

REGION Network 42: Error: Cooling fan doesn't come on
   RUNG wire#powerrail
      Contact( #HMI_VFD_Control.bSignalForward )
      Contact( #HMI_VFD_Control.bForwardOn )
      wire#w1
      I_Contact( #bInCoolingFan )
      { S7_Templates := "time_type := Time" } #TON_CoolingFan.TON(pt := T#30S, et => #tTemp)
      Coil( #bTON_CoolingFan )
   END_RUNG
   RUNG wire#powerrail
      Contact( #HMI_VFD_Control.bSignalReverse )
      Contact( #HMI_VFD_Control.bReverseOn )
   END_RUNG wire#w1
   // the same network as SCL:
   #TON_CoolingFan(IN := ((#HMI_VFD_Control.bSignalForward AND #HMI_VFD_Control.bForwardOn) OR (#HMI_VFD_Control.bSignalReverse AND #HMI_VFD_Control.bReverseOn)) AND NOT #bInCoolingFan,   // TON
                   PT := T#30S,
                   ET => #tTemp);
   #bTON_CoolingFan := #TON_CoolingFan.Q;
END_REGION

REGION Network 43: Error: No feedback from cooling fan
   RUNG wire#powerrail
      I_Contact( #bInEstop )
      Contact( #bTON_CoolingFan )
      I_Contact( #bInCoolingFan )
      S_Coil( #ERROR_VFD.NoCoolingFanFeedback )
   END_RUNG
   // the same network as SCL:
   IF NOT #bInEstop AND #bTON_CoolingFan AND NOT #bInCoolingFan THEN
       #ERROR_VFD.NoCoolingFanFeedback := TRUE;
   END_IF;
END_REGION

REGION Network 44: Scroll errors on the HMI
   // Call the Error-Scroller which cyles through all possible errors and checks 
   // their state for display on the HMI
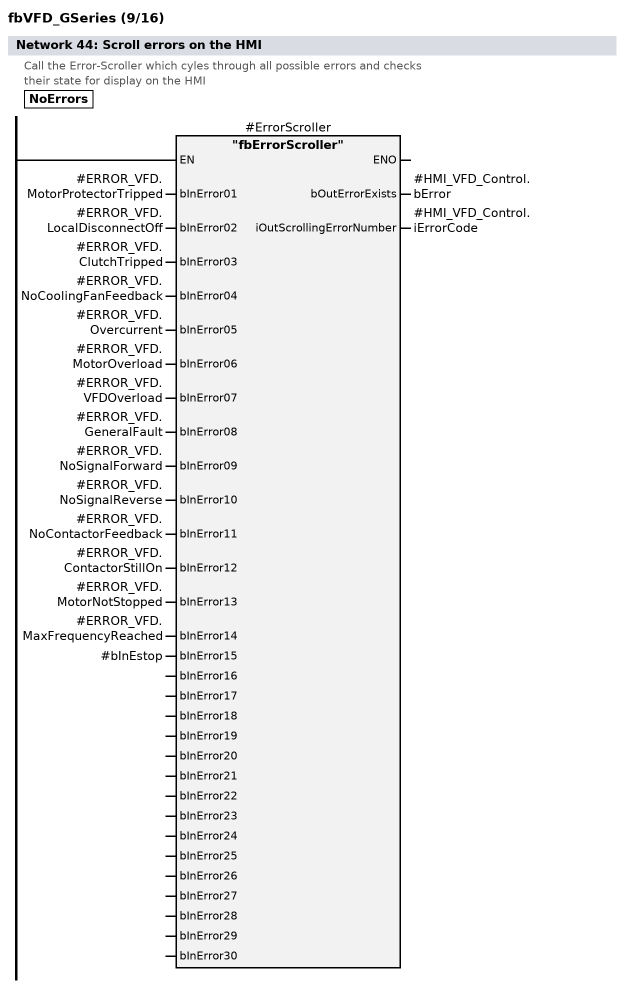
   Label( NoErrors )
   RUNG wire#powerrail
      #ErrorScroller(bInError01 := #ERROR_VFD.MotorProtectorTripped, bInError02 := #ERROR_VFD.LocalDisconnectOff, bInError03 := #ERROR_VFD.ClutchTripped, bInError04 := #ERROR_VFD.NoCoolingFanFeedback, bInError05 := #ERROR_VFD.Overcurrent, bInError06 := #ERROR_VFD.MotorOverload, bInError07 := #ERROR_VFD.VFDOverload, bInError08 := #ERROR_VFD.GeneralFault, bInError09 := #ERROR_VFD.NoSignalForward, bInError10 := #ERROR_VFD.NoSignalReverse, bInError11 := #ERROR_VFD.NoContactorFeedback, bInError12 := #ERROR_VFD.ContactorStillOn, bInError13 := #ERROR_VFD.MotorNotStopped, bInError14 := #ERROR_VFD.MaxFrequencyReached, bInError15 := #bInEstop, bInError16 :=, bInError17 :=, bInError18 :=, bInError19 :=, bInError20 :=, bInError21 :=, bInError22 :=, bInError23 :=, bInError24 :=, bInError25 :=, bInError26 :=, bInError27 :=, bInError28 :=, bInError29 :=, bInError30 :=, bOutErrorExists => #HMI_VFD_Control.bError, iOutScrollingErrorNumber => #HMI_VFD_Control.iErrorCode)
   END_RUNG
   // the same network as SCL:
   NoErrors:
   #ErrorScroller(bInError01 := #ERROR_VFD.MotorProtectorTripped,   // "fbErrorScroller"
                  bInError02 := #ERROR_VFD.LocalDisconnectOff,
                  bInError03 := #ERROR_VFD.ClutchTripped,
                  bInError04 := #ERROR_VFD.NoCoolingFanFeedback,
                  bInError05 := #ERROR_VFD.Overcurrent,
                  bInError06 := #ERROR_VFD.MotorOverload,
                  bInError07 := #ERROR_VFD.VFDOverload,
                  bInError08 := #ERROR_VFD.GeneralFault,
                  bInError09 := #ERROR_VFD.NoSignalForward,
                  bInError10 := #ERROR_VFD.NoSignalReverse,
                  bInError11 := #ERROR_VFD.NoContactorFeedback,
                  bInError12 := #ERROR_VFD.ContactorStillOn,
                  bInError13 := #ERROR_VFD.MotorNotStopped,
                  bInError14 := #ERROR_VFD.MaxFrequencyReached,
                  bInError15 := #bInEstop,
                  bOutErrorExists => #HMI_VFD_Control.bError,
                  iOutScrollingErrorNumber => #HMI_VFD_Control.iErrorCode);
END_REGION

REGION Network 45: Set major fault bit
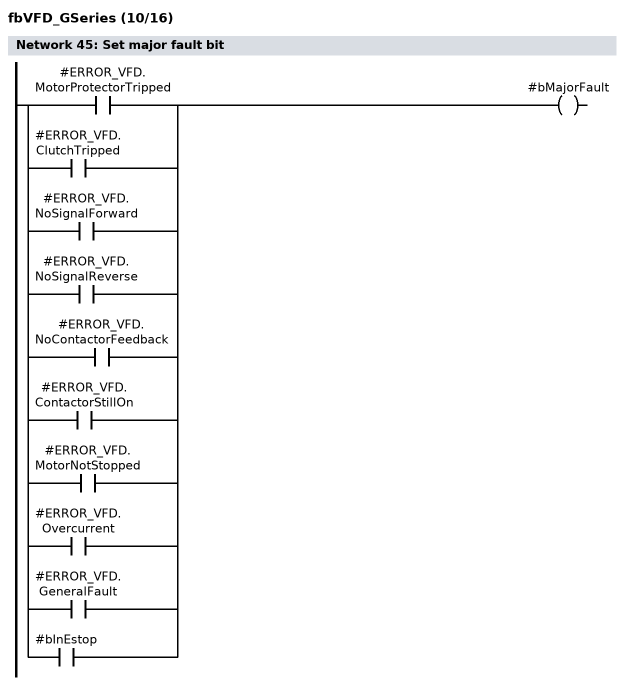
   RUNG wire#powerrail
      Contact( #ERROR_VFD.MotorProtectorTripped )
      wire#w1
      Coil( #bMajorFault )
   END_RUNG
   RUNG wire#powerrail
      Contact( #ERROR_VFD.ClutchTripped )
   END_RUNG wire#w1
   RUNG wire#powerrail
      Contact( #ERROR_VFD.NoSignalForward )
   END_RUNG wire#w1
   RUNG wire#powerrail
      Contact( #ERROR_VFD.NoSignalReverse )
   END_RUNG wire#w1
   RUNG wire#powerrail
      Contact( #ERROR_VFD.NoContactorFeedback )
   END_RUNG wire#w1
   RUNG wire#powerrail
      Contact( #ERROR_VFD.ContactorStillOn )
   END_RUNG wire#w1
   RUNG wire#powerrail
      Contact( #ERROR_VFD.MotorNotStopped )
   END_RUNG wire#w1
   RUNG wire#powerrail
      Contact( #ERROR_VFD.Overcurrent )
   END_RUNG wire#w1
   RUNG wire#powerrail
      Contact( #ERROR_VFD.GeneralFault )
   END_RUNG wire#w1
   RUNG wire#powerrail
      Contact( #bInEstop )
   END_RUNG wire#w1
   // the same network as SCL:
   #bMajorFault := #ERROR_VFD.MotorProtectorTripped OR #ERROR_VFD.ClutchTripped OR #ERROR_VFD.NoSignalForward OR #ERROR_VFD.NoSignalReverse OR #ERROR_VFD.NoContactorFeedback OR #ERROR_VFD.ContactorStillOn OR #ERROR_VFD.MotorNotStopped OR #ERROR_VFD.Overcurrent OR #ERROR_VFD.GeneralFault OR #bInEstop;
END_REGION

REGION Network 46: Set control bits based on major fault
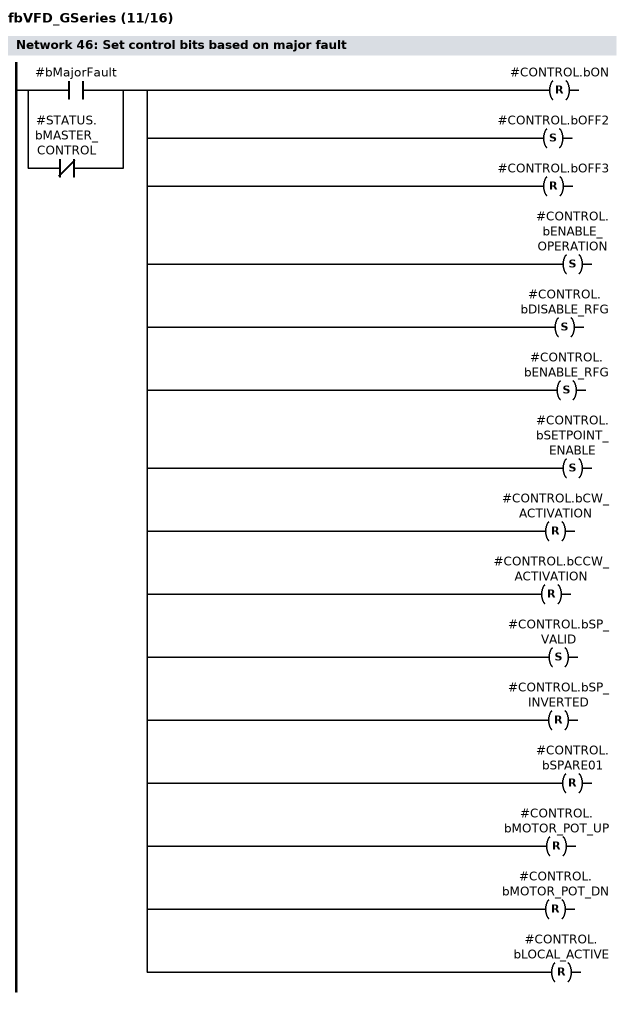
   RUNG wire#powerrail
      Contact( #bMajorFault )
      wire#w1
      R_Coil( #CONTROL.bON )
   END_RUNG
   RUNG wire#powerrail
      I_Contact( #STATUS.bMASTER_CONTROL )
   END_RUNG wire#w1
   RUNG wire#w1
      S_Coil( #CONTROL.bOFF2 )
   END_RUNG
   RUNG wire#w1
      R_Coil( #CONTROL.bOFF3 )
   END_RUNG
   RUNG wire#w1
      S_Coil( #CONTROL.bENABLE_OPERATION )
   END_RUNG
   RUNG wire#w1
      S_Coil( #CONTROL.bDISABLE_RFG )
   END_RUNG
   RUNG wire#w1
      S_Coil( #CONTROL.bENABLE_RFG )
   END_RUNG
   RUNG wire#w1
      S_Coil( #CONTROL.bSETPOINT_ENABLE )
   END_RUNG
   RUNG wire#w1
      R_Coil( #CONTROL.bCW_ACTIVATION )
   END_RUNG
   RUNG wire#w1
      R_Coil( #CONTROL.bCCW_ACTIVATION )
   END_RUNG
   RUNG wire#w1
      S_Coil( #CONTROL.bSP_VALID )
   END_RUNG
   RUNG wire#w1
      R_Coil( #CONTROL.bSP_INVERTED )
   END_RUNG
   RUNG wire#w1
      R_Coil( #CONTROL.bSPARE01 )
   END_RUNG
   RUNG wire#w1
      R_Coil( #CONTROL.bMOTOR_POT_UP )
   END_RUNG
   RUNG wire#w1
      R_Coil( #CONTROL.bMOTOR_POT_DN )
   END_RUNG
   RUNG wire#w1
      R_Coil( #CONTROL.bLOCAL_ACTIVE )
   END_RUNG
   // the same network as SCL:
   IF #bMajorFault OR NOT #STATUS.bMASTER_CONTROL THEN
       #CONTROL.bON := FALSE;
       #CONTROL.bOFF2 := TRUE;
       #CONTROL.bOFF3 := FALSE;
       #CONTROL.bENABLE_OPERATION := TRUE;
       #CONTROL.bDISABLE_RFG := TRUE;
       #CONTROL.bENABLE_RFG := TRUE;
       #CONTROL.bSETPOINT_ENABLE := TRUE;
       #CONTROL.bCW_ACTIVATION := FALSE;
       #CONTROL.bCCW_ACTIVATION := FALSE;
       #CONTROL.bSP_VALID := TRUE;
       #CONTROL.bSP_INVERTED := FALSE;
       #CONTROL.bSPARE01 := FALSE;
       #CONTROL.bMOTOR_POT_UP := FALSE;
       #CONTROL.bMOTOR_POT_DN := FALSE;
       #CONTROL.bLOCAL_ACTIVE := FALSE;
   END_IF;
END_REGION

REGION Network 47: Set control bits based on forward on command
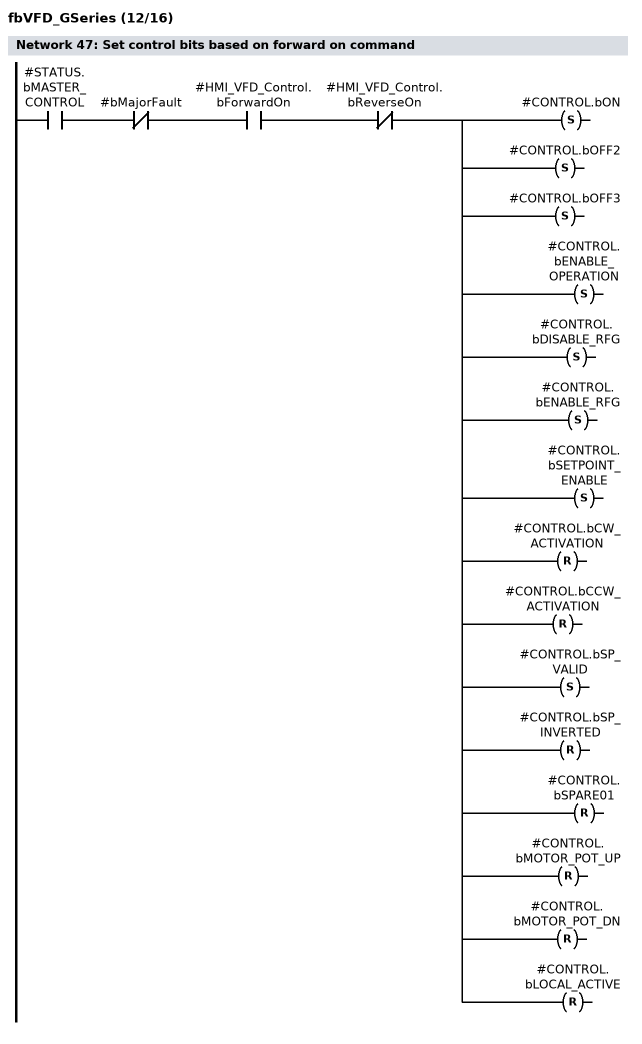
   RUNG wire#powerrail
      Contact( #STATUS.bMASTER_CONTROL )
      I_Contact( #bMajorFault )
      Contact( #HMI_VFD_Control.bForwardOn )
      I_Contact( #HMI_VFD_Control.bReverseOn )
      wire#w1
      S_Coil( #CONTROL.bON )
   END_RUNG
   RUNG wire#w1
      S_Coil( #CONTROL.bOFF2 )
   END_RUNG
   RUNG wire#w1
      S_Coil( #CONTROL.bOFF3 )
   END_RUNG
   RUNG wire#w1
      S_Coil( #CONTROL.bENABLE_OPERATION )
   END_RUNG
   RUNG wire#w1
      S_Coil( #CONTROL.bDISABLE_RFG )
   END_RUNG
   RUNG wire#w1
      S_Coil( #CONTROL.bENABLE_RFG )
   END_RUNG
   RUNG wire#w1
      S_Coil( #CONTROL.bSETPOINT_ENABLE )
   END_RUNG
   RUNG wire#w1
      R_Coil( #CONTROL.bCW_ACTIVATION )
   END_RUNG
   RUNG wire#w1
      R_Coil( #CONTROL.bCCW_ACTIVATION )
   END_RUNG
   RUNG wire#w1
      S_Coil( #CONTROL.bSP_VALID )
   END_RUNG
   RUNG wire#w1
      R_Coil( #CONTROL.bSP_INVERTED )
   END_RUNG
   RUNG wire#w1
      R_Coil( #CONTROL.bSPARE01 )
   END_RUNG
   RUNG wire#w1
      R_Coil( #CONTROL.bMOTOR_POT_UP )
   END_RUNG
   RUNG wire#w1
      R_Coil( #CONTROL.bMOTOR_POT_DN )
   END_RUNG
   RUNG wire#w1
      R_Coil( #CONTROL.bLOCAL_ACTIVE )
   END_RUNG
   // the same network as SCL:
   IF #STATUS.bMASTER_CONTROL AND NOT #bMajorFault AND #HMI_VFD_Control.bForwardOn AND NOT #HMI_VFD_Control.bReverseOn THEN
       #CONTROL.bON := TRUE;
       #CONTROL.bOFF2 := TRUE;
       #CONTROL.bOFF3 := TRUE;
       #CONTROL.bENABLE_OPERATION := TRUE;
       #CONTROL.bDISABLE_RFG := TRUE;
       #CONTROL.bENABLE_RFG := TRUE;
       #CONTROL.bSETPOINT_ENABLE := TRUE;
       #CONTROL.bCW_ACTIVATION := FALSE;
       #CONTROL.bCCW_ACTIVATION := FALSE;
       #CONTROL.bSP_VALID := TRUE;
       #CONTROL.bSP_INVERTED := FALSE;
       #CONTROL.bSPARE01 := FALSE;
       #CONTROL.bMOTOR_POT_UP := FALSE;
       #CONTROL.bMOTOR_POT_DN := FALSE;
       #CONTROL.bLOCAL_ACTIVE := FALSE;
   END_IF;
END_REGION

REGION Network 48: Set control bits based on Reverse on command
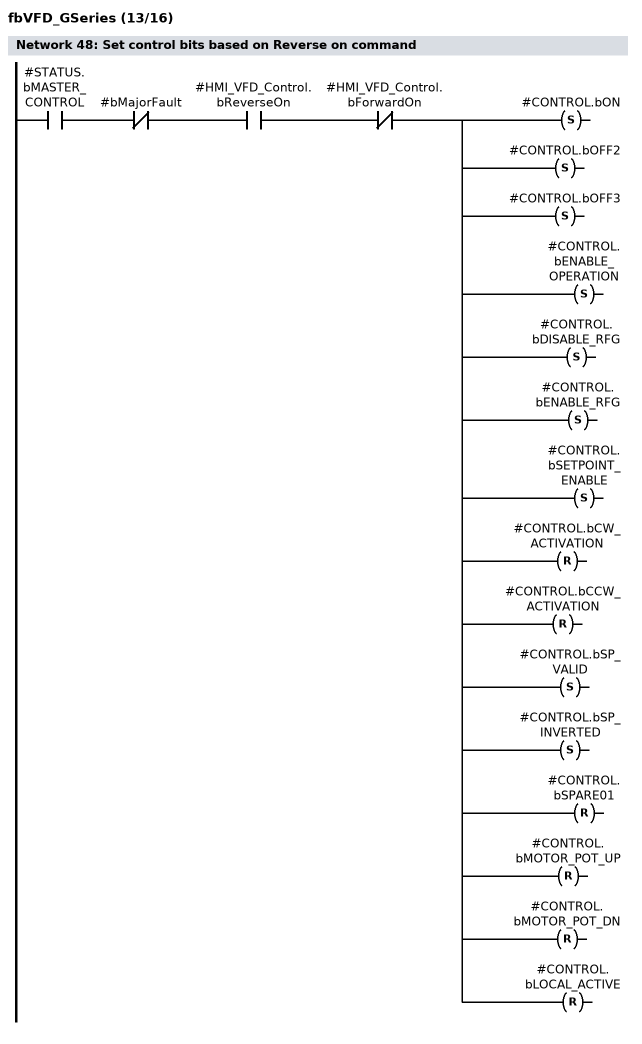
   RUNG wire#powerrail
      Contact( #STATUS.bMASTER_CONTROL )
      I_Contact( #bMajorFault )
      Contact( #HMI_VFD_Control.bReverseOn )
      I_Contact( #HMI_VFD_Control.bForwardOn )
      wire#w1
      S_Coil( #CONTROL.bON )
   END_RUNG
   RUNG wire#w1
      S_Coil( #CONTROL.bOFF2 )
   END_RUNG
   RUNG wire#w1
      S_Coil( #CONTROL.bOFF3 )
   END_RUNG
   RUNG wire#w1
      S_Coil( #CONTROL.bENABLE_OPERATION )
   END_RUNG
   RUNG wire#w1
      S_Coil( #CONTROL.bDISABLE_RFG )
   END_RUNG
   RUNG wire#w1
      S_Coil( #CONTROL.bENABLE_RFG )
   END_RUNG
   RUNG wire#w1
      S_Coil( #CONTROL.bSETPOINT_ENABLE )
   END_RUNG
   RUNG wire#w1
      R_Coil( #CONTROL.bCW_ACTIVATION )
   END_RUNG
   RUNG wire#w1
      R_Coil( #CONTROL.bCCW_ACTIVATION )
   END_RUNG
   RUNG wire#w1
      S_Coil( #CONTROL.bSP_VALID )
   END_RUNG
   RUNG wire#w1
      S_Coil( #CONTROL.bSP_INVERTED )
   END_RUNG
   RUNG wire#w1
      R_Coil( #CONTROL.bSPARE01 )
   END_RUNG
   RUNG wire#w1
      R_Coil( #CONTROL.bMOTOR_POT_UP )
   END_RUNG
   RUNG wire#w1
      R_Coil( #CONTROL.bMOTOR_POT_DN )
   END_RUNG
   RUNG wire#w1
      R_Coil( #CONTROL.bLOCAL_ACTIVE )
   END_RUNG
   // the same network as SCL:
   IF #STATUS.bMASTER_CONTROL AND NOT #bMajorFault AND #HMI_VFD_Control.bReverseOn AND NOT #HMI_VFD_Control.bForwardOn THEN
       #CONTROL.bON := TRUE;
       #CONTROL.bOFF2 := TRUE;
       #CONTROL.bOFF3 := TRUE;
       #CONTROL.bENABLE_OPERATION := TRUE;
       #CONTROL.bDISABLE_RFG := TRUE;
       #CONTROL.bENABLE_RFG := TRUE;
       #CONTROL.bSETPOINT_ENABLE := TRUE;
       #CONTROL.bCW_ACTIVATION := FALSE;
       #CONTROL.bCCW_ACTIVATION := FALSE;
       #CONTROL.bSP_VALID := TRUE;
       #CONTROL.bSP_INVERTED := TRUE;
       #CONTROL.bSPARE01 := FALSE;
       #CONTROL.bMOTOR_POT_UP := FALSE;
       #CONTROL.bMOTOR_POT_DN := FALSE;
       #CONTROL.bLOCAL_ACTIVE := FALSE;
   END_IF;
END_REGION

REGION Network 49: Set command bits when nothing is commanded, but no faults
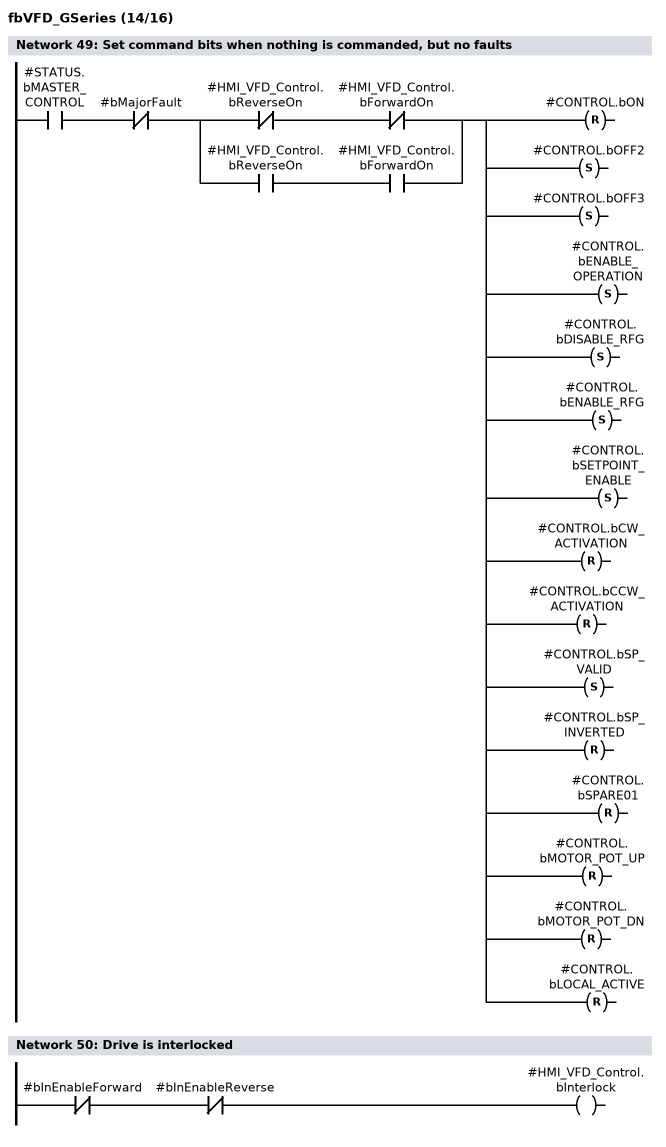
   RUNG wire#powerrail
      Contact( #STATUS.bMASTER_CONTROL )
      I_Contact( #bMajorFault )
      wire#w1
      I_Contact( #HMI_VFD_Control.bReverseOn )
      I_Contact( #HMI_VFD_Control.bForwardOn )
      wire#w2
      R_Coil( #CONTROL.bON )
   END_RUNG
   RUNG wire#w1
      Contact( #HMI_VFD_Control.bReverseOn )
      Contact( #HMI_VFD_Control.bForwardOn )
   END_RUNG wire#w2
   RUNG wire#w2
      S_Coil( #CONTROL.bOFF2 )
   END_RUNG
   RUNG wire#w2
      S_Coil( #CONTROL.bOFF3 )
   END_RUNG
   RUNG wire#w2
      S_Coil( #CONTROL.bENABLE_OPERATION )
   END_RUNG
   RUNG wire#w2
      S_Coil( #CONTROL.bDISABLE_RFG )
   END_RUNG
   RUNG wire#w2
      S_Coil( #CONTROL.bENABLE_RFG )
   END_RUNG
   RUNG wire#w2
      S_Coil( #CONTROL.bSETPOINT_ENABLE )
   END_RUNG
   RUNG wire#w2
      R_Coil( #CONTROL.bCW_ACTIVATION )
   END_RUNG
   RUNG wire#w2
      R_Coil( #CONTROL.bCCW_ACTIVATION )
   END_RUNG
   RUNG wire#w2
      S_Coil( #CONTROL.bSP_VALID )
   END_RUNG
   RUNG wire#w2
      R_Coil( #CONTROL.bSP_INVERTED )
   END_RUNG
   RUNG wire#w2
      R_Coil( #CONTROL.bSPARE01 )
   END_RUNG
   RUNG wire#w2
      R_Coil( #CONTROL.bMOTOR_POT_UP )
   END_RUNG
   RUNG wire#w2
      R_Coil( #CONTROL.bMOTOR_POT_DN )
   END_RUNG
   RUNG wire#w2
      R_Coil( #CONTROL.bLOCAL_ACTIVE )
   END_RUNG
   // the same network as SCL:
   IF #STATUS.bMASTER_CONTROL AND NOT #bMajorFault AND ((NOT #HMI_VFD_Control.bReverseOn AND NOT #HMI_VFD_Control.bForwardOn) OR (#HMI_VFD_Control.bReverseOn AND #HMI_VFD_Control.bForwardOn)) THEN
       #CONTROL.bON := FALSE;
       #CONTROL.bOFF2 := TRUE;
       #CONTROL.bOFF3 := TRUE;
       #CONTROL.bENABLE_OPERATION := TRUE;
       #CONTROL.bDISABLE_RFG := TRUE;
       #CONTROL.bENABLE_RFG := TRUE;
       #CONTROL.bSETPOINT_ENABLE := TRUE;
       #CONTROL.bCW_ACTIVATION := FALSE;
       #CONTROL.bCCW_ACTIVATION := FALSE;
       #CONTROL.bSP_VALID := TRUE;
       #CONTROL.bSP_INVERTED := FALSE;
       #CONTROL.bSPARE01 := FALSE;
       #CONTROL.bMOTOR_POT_UP := FALSE;
       #CONTROL.bMOTOR_POT_DN := FALSE;
       #CONTROL.bLOCAL_ACTIVE := FALSE;
   END_IF;
END_REGION

REGION Network 50: Drive is interlocked
   RUNG wire#powerrail
      I_Contact( #bInEnableForward )
      I_Contact( #bInEnableReverse )
      Coil( #HMI_VFD_Control.bInterlock )
   END_RUNG
   // the same network as SCL:
   #HMI_VFD_Control.bInterlock := NOT #bInEnableForward AND NOT #bInEnableReverse;
END_REGION

REGION Network 51: Set HMI status
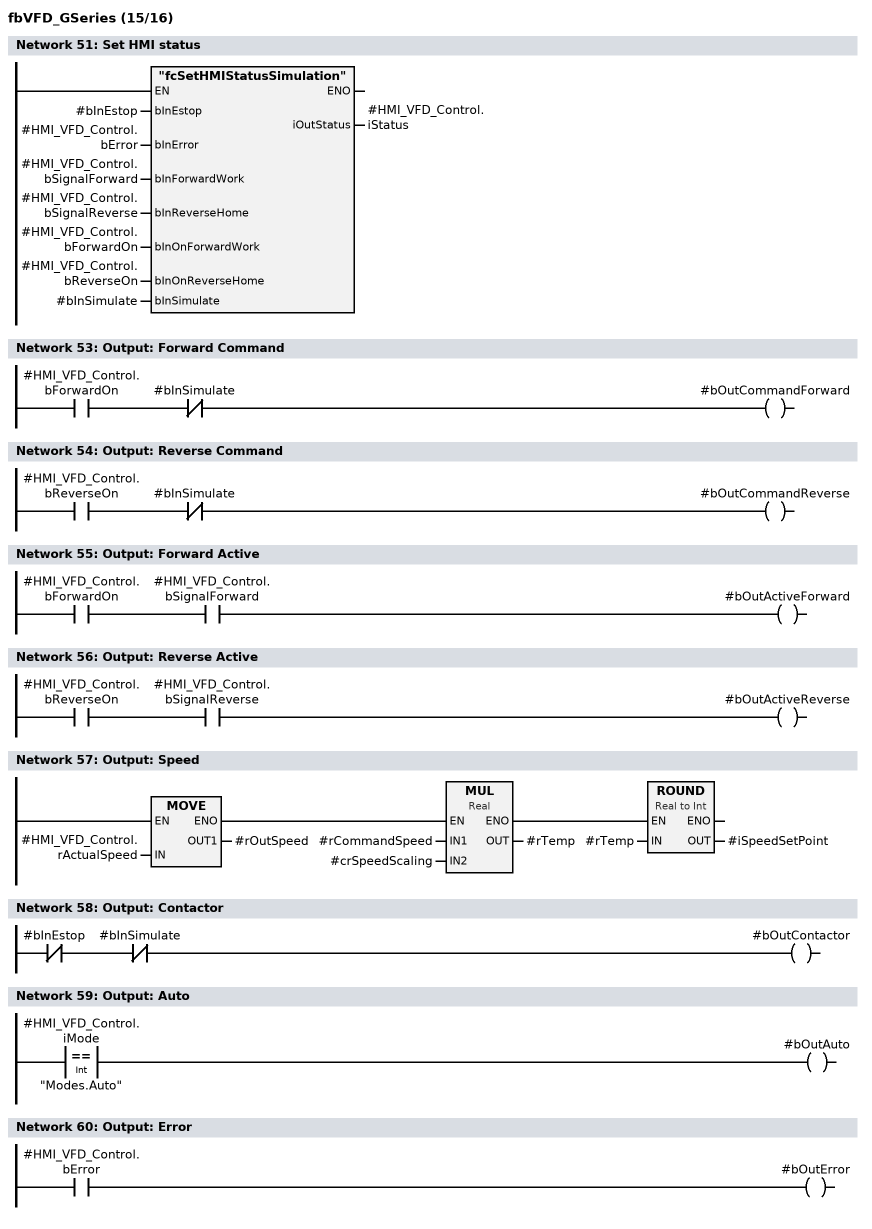
   RUNG wire#powerrail
      "fcSetHMIStatusSimulation"(bInEstop := #bInEstop, bInError := #HMI_VFD_Control.bError, bInForwardWork := #HMI_VFD_Control.bSignalForward, bInReverseHome := #HMI_VFD_Control.bSignalReverse, bInOnForwardWork := #HMI_VFD_Control.bForwardOn, bInOnReverseHome := #HMI_VFD_Control.bReverseOn, bInSimulate := #bInSimulate, iOutStatus => #HMI_VFD_Control.iStatus)
   END_RUNG
   // the same network as SCL:
   "fcSetHMIStatusSimulation"(bInEstop := #bInEstop,
                           bInError := #HMI_VFD_Control.bError,
                           bInForwardWork := #HMI_VFD_Control.bSignalForward,
                           bInReverseHome := #HMI_VFD_Control.bSignalReverse,
                           bInOnForwardWork := #HMI_VFD_Control.bForwardOn,
                           bInOnReverseHome := #HMI_VFD_Control.bReverseOn,
                           bInSimulate := #bInSimulate,
                           iOutStatus => #HMI_VFD_Control.iStatus);
END_REGION

REGION Network 52: --------------------------------------------------------- Outputs ------------------------------------------------------------------
END_REGION

REGION Network 53: Output: Forward Command
   RUNG wire#powerrail
      Contact( #HMI_VFD_Control.bForwardOn )
      I_Contact( #bInSimulate )
      Coil( #bOutCommandForward )
   END_RUNG
   // the same network as SCL:
   #bOutCommandForward := #HMI_VFD_Control.bForwardOn AND NOT #bInSimulate;
END_REGION

REGION Network 54: Output: Reverse Command
   RUNG wire#powerrail
      Contact( #HMI_VFD_Control.bReverseOn )
      I_Contact( #bInSimulate )
      Coil( #bOutCommandReverse )
   END_RUNG
   // the same network as SCL:
   #bOutCommandReverse := #HMI_VFD_Control.bReverseOn AND NOT #bInSimulate;
END_REGION

REGION Network 55: Output: Forward Active
   RUNG wire#powerrail
      Contact( #HMI_VFD_Control.bForwardOn )
      Contact( #HMI_VFD_Control.bSignalForward )
      Coil( #bOutActiveForward )
   END_RUNG
   // the same network as SCL:
   #bOutActiveForward := #HMI_VFD_Control.bForwardOn AND #HMI_VFD_Control.bSignalForward;
END_REGION

REGION Network 56: Output: Reverse Active
   RUNG wire#powerrail
      Contact( #HMI_VFD_Control.bReverseOn )
      Contact( #HMI_VFD_Control.bSignalReverse )
      Coil( #bOutActiveReverse )
   END_RUNG
   // the same network as SCL:
   #bOutActiveReverse := #HMI_VFD_Control.bReverseOn AND #HMI_VFD_Control.bSignalReverse;
END_REGION

REGION Network 57: Output: Speed
   RUNG wire#powerrail
      Move(in := #HMI_VFD_Control.rActualSpeed, out1 => #rOutSpeed)
      { S7_Templates := "SrcType := Real" } Mul(in1 := #rCommandSpeed, in2 := #crSpeedScaling, out => #rTemp)
      { S7_Templates := "[SrcType := Real, DestType := Int]" } Round(in := #rTemp, out => #iSpeedSetPoint)
   END_RUNG
   // the same network as SCL:
   #rOutSpeed := #HMI_VFD_Control.rActualSpeed;
   #rTemp := #rCommandSpeed * #crSpeedScaling;
   #iSpeedSetPoint := ROUND(#rTemp);
END_REGION

REGION Network 58: Output: Contactor
   RUNG wire#powerrail
      I_Contact( #bInEstop )
      I_Contact( #bInSimulate )
      Coil( #bOutContactor )
   END_RUNG
   // the same network as SCL:
   #bOutContactor := NOT #bInEstop AND NOT #bInSimulate;
END_REGION

REGION Network 59: Output: Auto
   RUNG wire#powerrail
      { S7_Templates := "SrcType := Int" } EQ_Contact(in1 := #HMI_VFD_Control.iMode, in2 := "Modes.Auto")
      Coil( #bOutAuto )
   END_RUNG
   // the same network as SCL:
   #bOutAuto := #HMI_VFD_Control.iMode = "Modes.Auto";
END_REGION

REGION Network 60: Output: Error
   RUNG wire#powerrail
      Contact( #HMI_VFD_Control.bError )
      Coil( #bOutError )
   END_RUNG
   // the same network as SCL:
   #bOutError := #HMI_VFD_Control.bError;
END_REGION

REGION Network 61: Output: Control Word
   // assemble control bits into control word
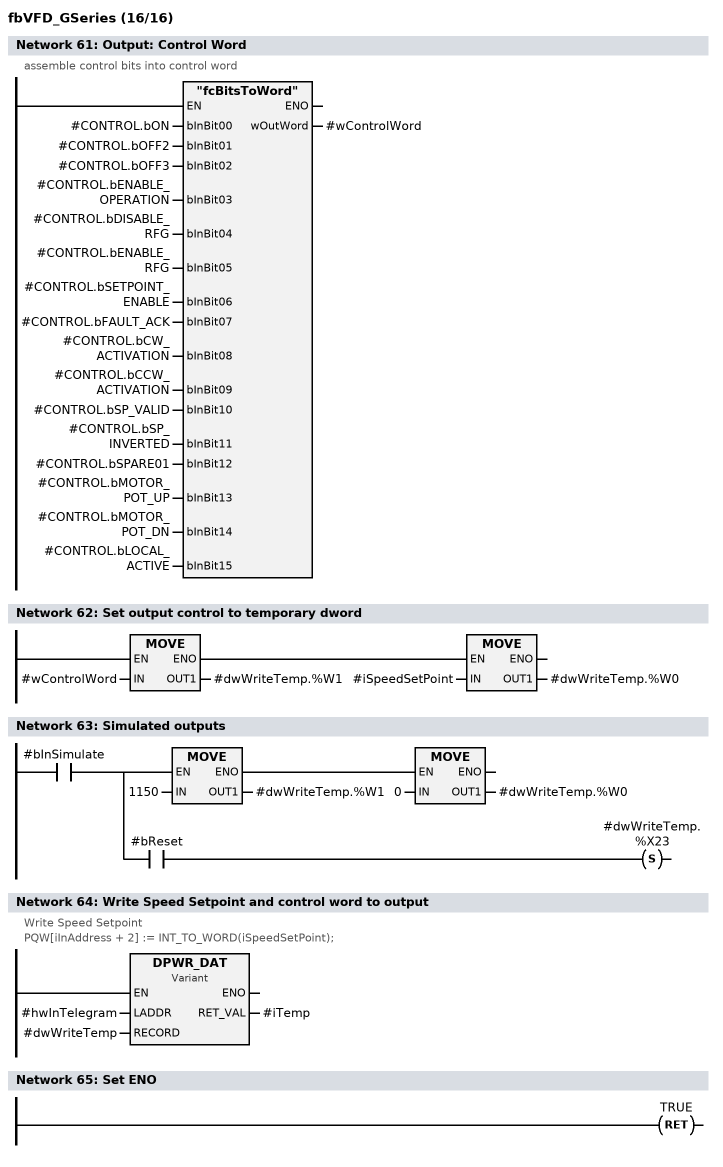
   RUNG wire#powerrail
      "fcBitsToWord"(bInBit00 := #CONTROL.bON, bInBit01 := #CONTROL.bOFF2, bInBit02 := #CONTROL.bOFF3, bInBit03 := #CONTROL.bENABLE_OPERATION, bInBit04 := #CONTROL.bDISABLE_RFG, bInBit05 := #CONTROL.bENABLE_RFG, bInBit06 := #CONTROL.bSETPOINT_ENABLE, bInBit07 := #CONTROL.bFAULT_ACK, bInBit08 := #CONTROL.bCW_ACTIVATION, bInBit09 := #CONTROL.bCCW_ACTIVATION, bInBit10 := #CONTROL.bSP_VALID, bInBit11 := #CONTROL.bSP_INVERTED, bInBit12 := #CONTROL.bSPARE01, bInBit13 := #CONTROL.bMOTOR_POT_UP, bInBit14 := #CONTROL.bMOTOR_POT_DN, bInBit15 := #CONTROL.bLOCAL_ACTIVE, wOutWord => #wControlWord)
   END_RUNG
   // the same network as SCL:
   "fcBitsToWord"(bInBit00 := #CONTROL.bON,
                  bInBit01 := #CONTROL.bOFF2,
                  bInBit02 := #CONTROL.bOFF3,
                  bInBit03 := #CONTROL.bENABLE_OPERATION,
                  bInBit04 := #CONTROL.bDISABLE_RFG,
                  bInBit05 := #CONTROL.bENABLE_RFG,
                  bInBit06 := #CONTROL.bSETPOINT_ENABLE,
                  bInBit07 := #CONTROL.bFAULT_ACK,
                  bInBit08 := #CONTROL.bCW_ACTIVATION,
                  bInBit09 := #CONTROL.bCCW_ACTIVATION,
                  bInBit10 := #CONTROL.bSP_VALID,
                  bInBit11 := #CONTROL.bSP_INVERTED,
                  bInBit12 := #CONTROL.bSPARE01,
                  bInBit13 := #CONTROL.bMOTOR_POT_UP,
                  bInBit14 := #CONTROL.bMOTOR_POT_DN,
                  bInBit15 := #CONTROL.bLOCAL_ACTIVE,
                  wOutWord => #wControlWord);
END_REGION

REGION Network 62: Set output control to temporary dword
   RUNG wire#powerrail
      Move(in := #wControlWord, out1 => #dwWriteTemp.%W1)
      Move(in := #iSpeedSetPoint, out1 => #dwWriteTemp.%W0)
   END_RUNG
   // the same network as SCL:
   #dwWriteTemp.%W1 := #wControlWord;
   #dwWriteTemp.%W0 := #iSpeedSetPoint;
END_REGION

REGION Network 63: Simulated outputs
   RUNG wire#powerrail
      Contact( #bInSimulate )
      wire#w1
      Move(in := 1150, out1 => #dwWriteTemp.%W1)
      Move(in := 0, out1 => #dwWriteTemp.%W0)
   END_RUNG
   RUNG wire#w1
      Contact( #bReset )
      S_Coil( #dwWriteTemp.%X23 )
   END_RUNG
   // the same network as SCL:
   IF #bInSimulate THEN
       #dwWriteTemp.%W1 := 1150;
       #dwWriteTemp.%W0 := 0;
   END_IF;
   IF #bInSimulate AND #bReset THEN #dwWriteTemp.%X23 := TRUE; END_IF;
END_REGION

REGION Network 64: Write Speed Setpoint and control word to output
   // Write Speed Setpoint
   // PQW[iInAddress + 2] := INT_TO_WORD(iSpeedSetPoint);
   RUNG wire#powerrail
      { S7_Templates := "[ptr_type := Variant, laddr_type := HW_IO]" } DPWR_DAT(LADDR := #hwInTelegram, RECORD := #dwWriteTemp, RET_VAL => #iTemp)
   END_RUNG
   // the same network as SCL:
   #iTemp := DPWR_DAT(LADDR := #hwInTelegram, RECORD := #dwWriteTemp);
END_REGION

REGION Network 65: Set ENO
   RUNG wire#powerrail
      ReturnCoil( TRUE )
   END_RUNG
   // the same network as SCL:
   ENO := TRUE;
   RETURN;
END_REGION
END_FUNCTION_BLOCK

FUNCTION "fcHMIBitEnable" : Void   // FC329, LAD
TITLE = Handles an async reading of an HMI bit to avoid race conditions, includes an enable bit
{ S7_Optimized_Access := 'TRUE' }
VERSION : 0.1
// stored: AutoNumber true, IsIECCheckEnabled false, SetENOAutomatically false, UDAEnableTagReadback false
   VAR_INPUT
      bInToggle : Bool;
      bInLatch : Bool;
      bInEnable : Bool;
   END_VAR
   VAR_OUTPUT
      bOutEnable : Bool;
   END_VAR
   VAR_IN_OUT
      bInOutHMI : Bool;
      bInOutPLC : Bool;
   END_VAR
   VAR_TEMP   // added for the SCL form of the ladder/FBD networks
      _w1 : Bool;
   END_VAR
BEGIN

REGION Network 1: If not latching or toggling, reset the PLC bit every scan
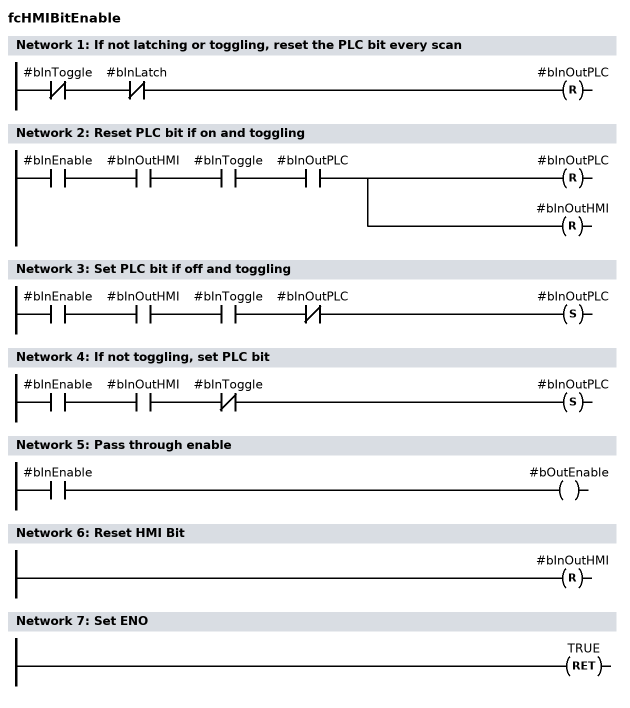
   RUNG wire#powerrail
      I_Contact( #bInToggle )
      I_Contact( #bInLatch )
      R_Coil( #bInOutPLC )
   END_RUNG
   // the same network as SCL:
   IF NOT #bInToggle AND NOT #bInLatch THEN #bInOutPLC := FALSE; END_IF;
END_REGION

REGION Network 2: Reset PLC bit if on and toggling
   RUNG wire#powerrail
      Contact( #bInEnable )
      Contact( #bInOutHMI )
      Contact( #bInToggle )
      Contact( #bInOutPLC )
      wire#w1
      R_Coil( #bInOutPLC )
   END_RUNG
   RUNG wire#w1
      R_Coil( #bInOutHMI )
   END_RUNG
   // the same network as SCL:
   #_w1 := #bInEnable AND #bInOutHMI AND #bInToggle AND #bInOutPLC;
   IF #_w1 THEN
       #bInOutPLC := FALSE;
       #bInOutHMI := FALSE;
   END_IF;
END_REGION

REGION Network 3: Set PLC bit if off and toggling
   RUNG wire#powerrail
      Contact( #bInEnable )
      Contact( #bInOutHMI )
      Contact( #bInToggle )
      I_Contact( #bInOutPLC )
      S_Coil( #bInOutPLC )
   END_RUNG
   // the same network as SCL:
   IF #bInEnable AND #bInOutHMI AND #bInToggle AND NOT #bInOutPLC THEN #bInOutPLC := TRUE; END_IF;
END_REGION

REGION Network 4: If not toggling, set PLC bit
   RUNG wire#powerrail
      Contact( #bInEnable )
      Contact( #bInOutHMI )
      I_Contact( #bInToggle )
      S_Coil( #bInOutPLC )
   END_RUNG
   // the same network as SCL:
   IF #bInEnable AND #bInOutHMI AND NOT #bInToggle THEN #bInOutPLC := TRUE; END_IF;
END_REGION

REGION Network 5: Pass through enable
   RUNG wire#powerrail
      Contact( #bInEnable )
      Coil( #bOutEnable )
   END_RUNG
   // the same network as SCL:
   #bOutEnable := #bInEnable;
END_REGION

REGION Network 6: Reset HMI Bit
   RUNG wire#powerrail
      R_Coil( #bInOutHMI )
   END_RUNG
   // the same network as SCL:
   #bInOutHMI := FALSE;
END_REGION

REGION Network 7: Set ENO
   RUNG wire#powerrail
      ReturnCoil( TRUE )
   END_RUNG
   // the same network as SCL:
   ENO := TRUE;
   RETURN;
END_REGION
END_FUNCTION

FUNCTION "fcWordToBits" : Void   // FC303, LAD
TITLE = Breaks A Word Into Individual Bits
{ S7_Optimized_Access := 'TRUE' }
AUTHOR : DMC
FAMILY : LowLevel
VERSION : 0.1
// stored: AutoNumber false, IsIECCheckEnabled false, SetENOAutomatically false, UDAEnableTagReadback false
   VAR_INPUT
      wInWord : Word;   // Word to be broken into individual bits
   END_VAR
   VAR_OUTPUT
      bOutBit00 : Bool;   // Bit 0
      bOutBit01 : Bool;   // Bit 1
      bOutBit02 : Bool;   // Bit 2
      bOutBit03 : Bool;   // Bit 3
      bOutBit04 : Bool;   // Bit 4
      bOutBit05 : Bool;   // Bit 5
      bOutBit06 : Bool;   // Bit 6
      bOutBit07 : Bool;   // Bit 7
      bOutBit08 : Bool;   // Bit 8
      bOutBit09 : Bool;   // Bit 9
      bOutBit10 : Bool;   // Bit 10
      bOutBit11 : Bool;   // Bit 11
      bOutBit12 : Bool;   // Bit 12
      bOutBit13 : Bool;   // Bit 13
      bOutBit14 : Bool;   // Bit 14
      bOutBit15 : Bool;   // Bit 15
   END_VAR
BEGIN

REGION Network 1: Bit0
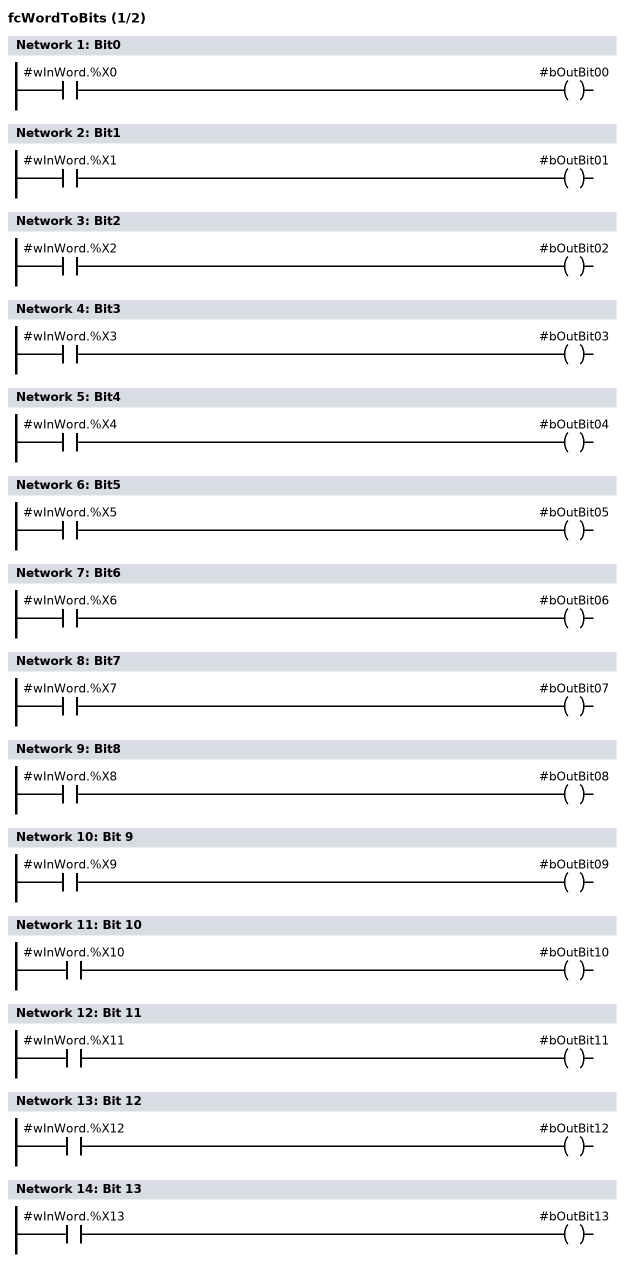
   RUNG wire#powerrail
      Contact( #wInWord.%X0 )
      Coil( #bOutBit00 )
   END_RUNG
   // the same network as SCL:
   #bOutBit00 := #wInWord.%X0;
END_REGION

REGION Network 2: Bit1
   RUNG wire#powerrail
      Contact( #wInWord.%X1 )
      Coil( #bOutBit01 )
   END_RUNG
   // the same network as SCL:
   #bOutBit01 := #wInWord.%X1;
END_REGION

REGION Network 3: Bit2
   RUNG wire#powerrail
      Contact( #wInWord.%X2 )
      Coil( #bOutBit02 )
   END_RUNG
   // the same network as SCL:
   #bOutBit02 := #wInWord.%X2;
END_REGION

REGION Network 4: Bit3
   RUNG wire#powerrail
      Contact( #wInWord.%X3 )
      Coil( #bOutBit03 )
   END_RUNG
   // the same network as SCL:
   #bOutBit03 := #wInWord.%X3;
END_REGION

REGION Network 5: Bit4
   RUNG wire#powerrail
      Contact( #wInWord.%X4 )
      Coil( #bOutBit04 )
   END_RUNG
   // the same network as SCL:
   #bOutBit04 := #wInWord.%X4;
END_REGION

REGION Network 6: Bit5
   RUNG wire#powerrail
      Contact( #wInWord.%X5 )
      Coil( #bOutBit05 )
   END_RUNG
   // the same network as SCL:
   #bOutBit05 := #wInWord.%X5;
END_REGION

REGION Network 7: Bit6
   RUNG wire#powerrail
      Contact( #wInWord.%X6 )
      Coil( #bOutBit06 )
   END_RUNG
   // the same network as SCL:
   #bOutBit06 := #wInWord.%X6;
END_REGION

REGION Network 8: Bit7
   RUNG wire#powerrail
      Contact( #wInWord.%X7 )
      Coil( #bOutBit07 )
   END_RUNG
   // the same network as SCL:
   #bOutBit07 := #wInWord.%X7;
END_REGION

REGION Network 9: Bit8
   RUNG wire#powerrail
      Contact( #wInWord.%X8 )
      Coil( #bOutBit08 )
   END_RUNG
   // the same network as SCL:
   #bOutBit08 := #wInWord.%X8;
END_REGION

REGION Network 10: Bit 9
   RUNG wire#powerrail
      Contact( #wInWord.%X9 )
      Coil( #bOutBit09 )
   END_RUNG
   // the same network as SCL:
   #bOutBit09 := #wInWord.%X9;
END_REGION

REGION Network 11: Bit 10
   RUNG wire#powerrail
      Contact( #wInWord.%X10 )
      Coil( #bOutBit10 )
   END_RUNG
   // the same network as SCL:
   #bOutBit10 := #wInWord.%X10;
END_REGION

REGION Network 12: Bit 11
   RUNG wire#powerrail
      Contact( #wInWord.%X11 )
      Coil( #bOutBit11 )
   END_RUNG
   // the same network as SCL:
   #bOutBit11 := #wInWord.%X11;
END_REGION

REGION Network 13: Bit 12
   RUNG wire#powerrail
      Contact( #wInWord.%X12 )
      Coil( #bOutBit12 )
   END_RUNG
   // the same network as SCL:
   #bOutBit12 := #wInWord.%X12;
END_REGION

REGION Network 14: Bit 13
   RUNG wire#powerrail
      Contact( #wInWord.%X13 )
      Coil( #bOutBit13 )
   END_RUNG
   // the same network as SCL:
   #bOutBit13 := #wInWord.%X13;
END_REGION

REGION Network 15: Bit 14
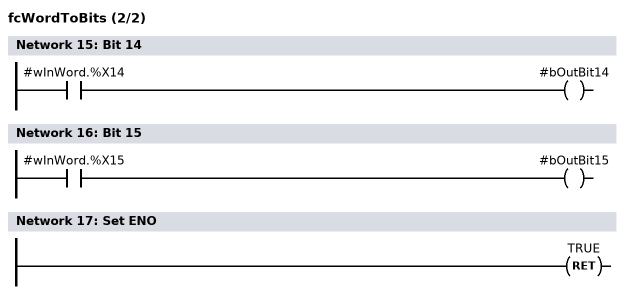
   RUNG wire#powerrail
      Contact( #wInWord.%X14 )
      Coil( #bOutBit14 )
   END_RUNG
   // the same network as SCL:
   #bOutBit14 := #wInWord.%X14;
END_REGION

REGION Network 16: Bit 15
   RUNG wire#powerrail
      Contact( #wInWord.%X15 )
      Coil( #bOutBit15 )
   END_RUNG
   // the same network as SCL:
   #bOutBit15 := #wInWord.%X15;
END_REGION

REGION Network 17: Set ENO
   RUNG wire#powerrail
      ReturnCoil( TRUE )
   END_RUNG
   // the same network as SCL:
   ENO := TRUE;
   RETURN;
END_REGION
END_FUNCTION

FUNCTION_BLOCK "fbErrorScroller"   // FB330, LAD
TITLE = Scrolls through the error codes for display on the HMI
{ S7_Optimized_Access := 'TRUE' }
AUTHOR : DMC
FAMILY : Error
VERSION : 0.1
// stored: AutoNumber false, IsIECCheckEnabled false, IsRetainMemResEnabled false, MemoryReserve 100, SetENOAutomatically false, UDAEnableTagReadback false
   VAR_INPUT
      bInError01 { ExternalAccessible := 'False'; ExternalVisible := 'False'; ExternalWritable := 'False'} : Bool;   // Error 1 In Error Array
      bInError02 { ExternalAccessible := 'False'; ExternalVisible := 'False'; ExternalWritable := 'False'} : Bool;   // Error 2 In Error Array
      bInError03 { ExternalAccessible := 'False'; ExternalVisible := 'False'; ExternalWritable := 'False'} : Bool;   // Error 3 In Error Array
      bInError04 { ExternalAccessible := 'False'; ExternalVisible := 'False'; ExternalWritable := 'False'} : Bool;   // Error 4 In Error Array
      bInError05 { ExternalAccessible := 'False'; ExternalVisible := 'False'; ExternalWritable := 'False'} : Bool;   // Error 5 In Error Array
      bInError06 { ExternalAccessible := 'False'; ExternalVisible := 'False'; ExternalWritable := 'False'} : Bool;   // Error 6 In Error Array
      bInError07 { ExternalAccessible := 'False'; ExternalVisible := 'False'; ExternalWritable := 'False'} : Bool;   // Error 7 In Error Array
      bInError08 { ExternalAccessible := 'False'; ExternalVisible := 'False'; ExternalWritable := 'False'} : Bool;   // Error 8 In Error Array
      bInError09 { ExternalAccessible := 'False'; ExternalVisible := 'False'; ExternalWritable := 'False'} : Bool;   // Error 9 In Error Array
      bInError10 { ExternalAccessible := 'False'; ExternalVisible := 'False'; ExternalWritable := 'False'} : Bool;   // Error 10 In Error Array
      bInError11 { ExternalAccessible := 'False'; ExternalVisible := 'False'; ExternalWritable := 'False'} : Bool;   // Error 11 In Error Array
      bInError12 { ExternalAccessible := 'False'; ExternalVisible := 'False'; ExternalWritable := 'False'} : Bool;   // Error 12 In Error Array
      bInError13 { ExternalAccessible := 'False'; ExternalVisible := 'False'; ExternalWritable := 'False'} : Bool;   // Error 13 In Error Array
      bInError14 { ExternalAccessible := 'False'; ExternalVisible := 'False'; ExternalWritable := 'False'} : Bool;   // Error 14 In Error Array
      bInError15 { ExternalAccessible := 'False'; ExternalVisible := 'False'; ExternalWritable := 'False'} : Bool;   // Error 15 In Error Array
      bInError16 { ExternalAccessible := 'False'; ExternalVisible := 'False'; ExternalWritable := 'False'} : Bool;   // Error 16 In Error Array
      bInError17 { ExternalAccessible := 'False'; ExternalVisible := 'False'; ExternalWritable := 'False'} : Bool;   // Error 17 In Error Array
      bInError18 { ExternalAccessible := 'False'; ExternalVisible := 'False'; ExternalWritable := 'False'} : Bool;   // Error 18 In Error Array
      bInError19 { ExternalAccessible := 'False'; ExternalVisible := 'False'; ExternalWritable := 'False'} : Bool;   // Error 19 In Error Array
      bInError20 { ExternalAccessible := 'False'; ExternalVisible := 'False'; ExternalWritable := 'False'} : Bool;   // Error 20 In Error Array
      bInError21 { ExternalAccessible := 'False'; ExternalVisible := 'False'; ExternalWritable := 'False'} : Bool;   // Error 21 In Error Array
      bInError22 { ExternalAccessible := 'False'; ExternalVisible := 'False'; ExternalWritable := 'False'} : Bool;   // Error 22 In Error Array
      bInError23 { ExternalAccessible := 'False'; ExternalVisible := 'False'; ExternalWritable := 'False'} : Bool;   // Error 23 In Error Array
      bInError24 { ExternalAccessible := 'False'; ExternalVisible := 'False'; ExternalWritable := 'False'} : Bool;   // Error 24 In Error Array
      bInError25 { ExternalAccessible := 'False'; ExternalVisible := 'False'; ExternalWritable := 'False'} : Bool;   // Error 25 In Error Array
      bInError26 { ExternalAccessible := 'False'; ExternalVisible := 'False'; ExternalWritable := 'False'} : Bool;   // Error 26 In Error Array
      bInError27 { ExternalAccessible := 'False'; ExternalVisible := 'False'; ExternalWritable := 'False'} : Bool;   // Error 27 In Error Array
      bInError28 { ExternalAccessible := 'False'; ExternalVisible := 'False'; ExternalWritable := 'False'} : Bool;   // Error 28 In Error Array
      bInError29 { ExternalAccessible := 'False'; ExternalVisible := 'False'; ExternalWritable := 'False'} : Bool;   // Error 29 In Error Array
      bInError30 { ExternalAccessible := 'False'; ExternalVisible := 'False'; ExternalWritable := 'False'} : Bool;   // Error 30 In Error Array
   END_VAR
   VAR_OUTPUT
      bOutErrorExists { ExternalAccessible := 'False'; ExternalVisible := 'False'; ExternalWritable := 'False'} : Bool;   // An Error Exists
      iOutScrollingErrorNumber { ExternalAccessible := 'False'; ExternalVisible := 'False'; ExternalWritable := 'False'} : Int;   // Current Index when scrolling through errors
   END_VAR
   VAR
      TON_ErrorDelay { ExternalAccessible := 'False'; ExternalVisible := 'False'; ExternalWritable := 'False'; S7_SetPoint := 'True'} : TON_TIME;   // Delay between each scroll for a new error
   END_VAR
   VAR DB_SPECIFIC
      abErrors { ExternalAccessible := 'False'; ExternalVisible := 'False'; ExternalWritable := 'False'} : Array[#ciIndexLow..#ciIndexHigh] of Bool;
   END_VAR
   VAR
      iNextScrollNum { ExternalAccessible := 'False'; ExternalVisible := 'False'; ExternalWritable := 'False'} : Int := 1;   // Index of next error position
      iErrorsScrollNum { ExternalAccessible := 'False'; ExternalVisible := 'False'; ExternalWritable := 'False'} : Int := 1;   // Index of current error position
      bScrolling { ExternalAccessible := 'False'; ExternalVisible := 'False'; ExternalWritable := 'False'} : Bool;   // Indicates we are scrolling
      bTON_ErrorDelay { ExternalAccessible := 'False'; ExternalVisible := 'False'; ExternalWritable := 'False'} : Bool;
   END_VAR
   VAR_TEMP
      bErrorExists : Bool;   // Error Exists
   END_VAR
   VAR CONSTANT
      ciNoErrrors : Int := 0;
      ciIndexLow : Int := 1;
      ciIndexHigh : Int := 30;
   END_VAR
   VAR_TEMP   // added for the SCL form of the ladder/FBD networks
      _w1 : Bool;
   END_VAR
BEGIN

REGION Network 1: Check for valid array indexes
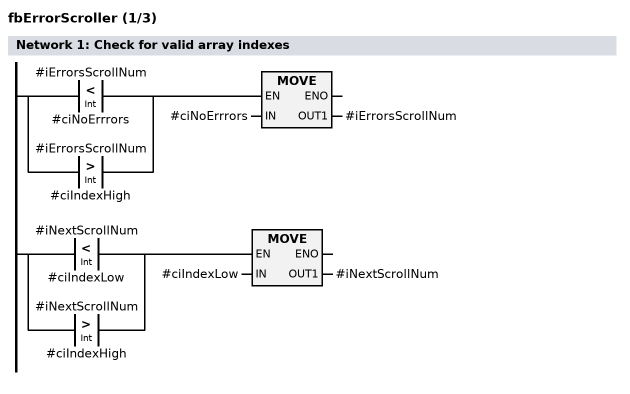
   RUNG wire#powerrail
      { S7_Templates := "SrcType := Int" } LT_Contact(in1 := #iErrorsScrollNum, in2 := #ciNoErrrors)
      wire#w1
      Move(in := #ciNoErrrors, out1 => #iErrorsScrollNum)
   END_RUNG
   RUNG wire#powerrail
      { S7_Templates := "SrcType := Int" } GT_Contact(in1 := #iErrorsScrollNum, in2 := #ciIndexHigh)
   END_RUNG wire#w1
   RUNG wire#powerrail
      { S7_Templates := "SrcType := Int" } LT_Contact(in1 := #iNextScrollNum, in2 := #ciIndexLow)
      wire#w2
      Move(in := #ciIndexLow, out1 => #iNextScrollNum)
   END_RUNG
   RUNG wire#powerrail
      { S7_Templates := "SrcType := Int" } GT_Contact(in1 := #iNextScrollNum, in2 := #ciIndexHigh)
   END_RUNG wire#w2
   // the same network as SCL:
   IF (#iErrorsScrollNum < #ciNoErrrors) OR (#iErrorsScrollNum > #ciIndexHigh) THEN
       #iErrorsScrollNum := #ciNoErrrors;
   END_IF;
   IF (#iNextScrollNum < #ciIndexLow) OR (#iNextScrollNum > #ciIndexHigh) THEN
       #iNextScrollNum := #ciIndexLow;
   END_IF;
END_REGION

REGION Network 2: Check if error exists
   // OR all of the possible errors. If any error Exists, SET bErrorExists
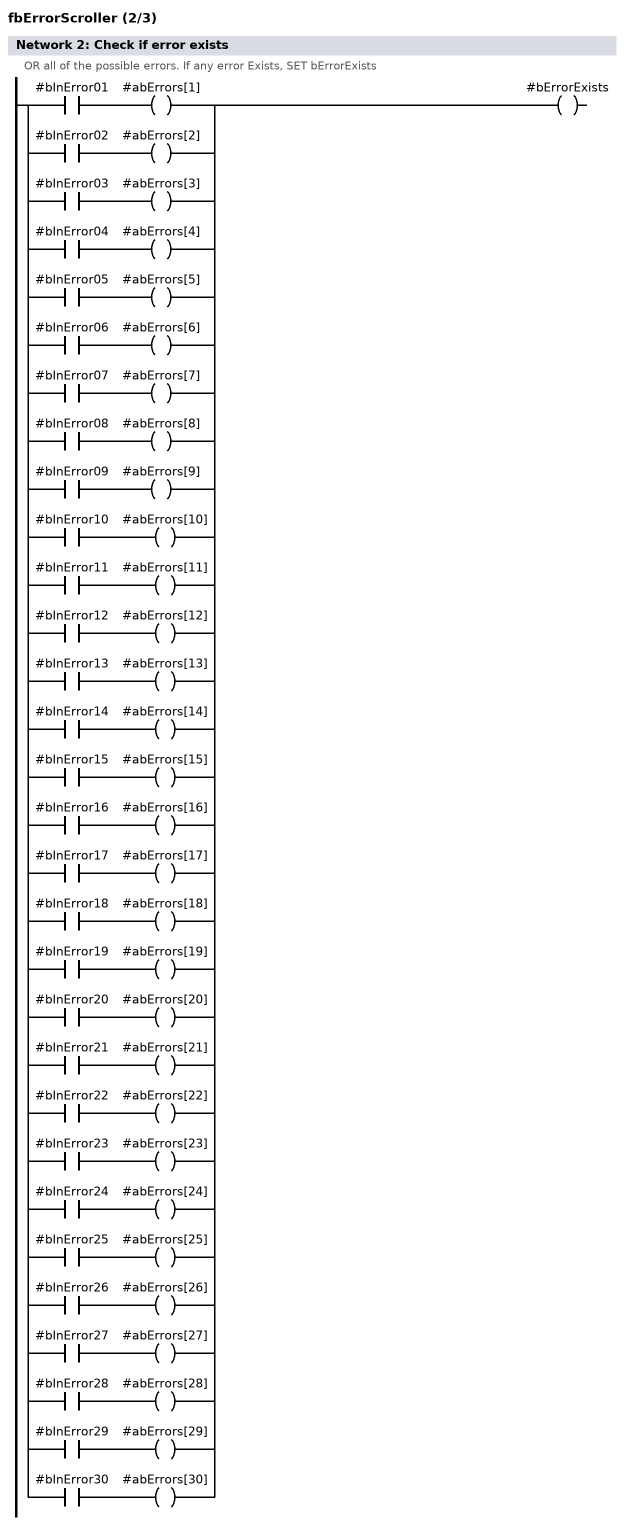
   RUNG wire#powerrail
      Contact( #bInError01 )
      Coil( #abErrors[1] )
      wire#w1
      Coil( #bErrorExists )
   END_RUNG
   RUNG wire#powerrail
      Contact( #bInError02 )
      Coil( #abErrors[2] )
   END_RUNG wire#w1
   RUNG wire#powerrail
      Contact( #bInError03 )
      Coil( #abErrors[3] )
   END_RUNG wire#w1
   RUNG wire#powerrail
      Contact( #bInError04 )
      Coil( #abErrors[4] )
   END_RUNG wire#w1
   RUNG wire#powerrail
      Contact( #bInError05 )
      Coil( #abErrors[5] )
   END_RUNG wire#w1
   RUNG wire#powerrail
      Contact( #bInError06 )
      Coil( #abErrors[6] )
   END_RUNG wire#w1
   RUNG wire#powerrail
      Contact( #bInError07 )
      Coil( #abErrors[7] )
   END_RUNG wire#w1
   RUNG wire#powerrail
      Contact( #bInError08 )
      Coil( #abErrors[8] )
   END_RUNG wire#w1
   RUNG wire#powerrail
      Contact( #bInError09 )
      Coil( #abErrors[9] )
   END_RUNG wire#w1
   RUNG wire#powerrail
      Contact( #bInError10 )
      Coil( #abErrors[10] )
   END_RUNG wire#w1
   RUNG wire#powerrail
      Contact( #bInError11 )
      Coil( #abErrors[11] )
   END_RUNG wire#w1
   RUNG wire#powerrail
      Contact( #bInError12 )
      Coil( #abErrors[12] )
   END_RUNG wire#w1
   RUNG wire#powerrail
      Contact( #bInError13 )
      Coil( #abErrors[13] )
   END_RUNG wire#w1
   RUNG wire#powerrail
      Contact( #bInError14 )
      Coil( #abErrors[14] )
   END_RUNG wire#w1
   RUNG wire#powerrail
      Contact( #bInError15 )
      Coil( #abErrors[15] )
   END_RUNG wire#w1
   RUNG wire#powerrail
      Contact( #bInError16 )
      Coil( #abErrors[16] )
   END_RUNG wire#w1
   RUNG wire#powerrail
      Contact( #bInError17 )
      Coil( #abErrors[17] )
   END_RUNG wire#w1
   RUNG wire#powerrail
      Contact( #bInError18 )
      Coil( #abErrors[18] )
   END_RUNG wire#w1
   RUNG wire#powerrail
      Contact( #bInError19 )
      Coil( #abErrors[19] )
   END_RUNG wire#w1
   RUNG wire#powerrail
      Contact( #bInError20 )
      Coil( #abErrors[20] )
   END_RUNG wire#w1
   RUNG wire#powerrail
      Contact( #bInError21 )
      Coil( #abErrors[21] )
   END_RUNG wire#w1
   RUNG wire#powerrail
      Contact( #bInError22 )
      Coil( #abErrors[22] )
   END_RUNG wire#w1
   RUNG wire#powerrail
      Contact( #bInError23 )
      Coil( #abErrors[23] )
   END_RUNG wire#w1
   RUNG wire#powerrail
      Contact( #bInError24 )
      Coil( #abErrors[24] )
   END_RUNG wire#w1
   RUNG wire#powerrail
      Contact( #bInError25 )
      Coil( #abErrors[25] )
   END_RUNG wire#w1
   RUNG wire#powerrail
      Contact( #bInError26 )
      Coil( #abErrors[26] )
   END_RUNG wire#w1
   RUNG wire#powerrail
      Contact( #bInError27 )
      Coil( #abErrors[27] )
   END_RUNG wire#w1
   RUNG wire#powerrail
      Contact( #bInError28 )
      Coil( #abErrors[28] )
   END_RUNG wire#w1
   RUNG wire#powerrail
      Contact( #bInError29 )
      Coil( #abErrors[29] )
   END_RUNG wire#w1
   RUNG wire#powerrail
      Contact( #bInError30 )
      Coil( #abErrors[30] )
   END_RUNG wire#w1
   // the same network as SCL:
   #abErrors[1] := #bInError01;
   #abErrors[2] := #bInError02;
   #abErrors[3] := #bInError03;
   #abErrors[4] := #bInError04;
   #abErrors[5] := #bInError05;
   #abErrors[6] := #bInError06;
   #abErrors[7] := #bInError07;
   #abErrors[8] := #bInError08;
   #abErrors[9] := #bInError09;
   #abErrors[10] := #bInError10;
   #abErrors[11] := #bInError11;
   #abErrors[12] := #bInError12;
   #abErrors[13] := #bInError13;
   #abErrors[14] := #bInError14;
   #abErrors[15] := #bInError15;
   #abErrors[16] := #bInError16;
   #abErrors[17] := #bInError17;
   #abErrors[18] := #bInError18;
   #abErrors[19] := #bInError19;
   #abErrors[20] := #bInError20;
   #abErrors[21] := #bInError21;
   #abErrors[22] := #bInError22;
   #abErrors[23] := #bInError23;
   #abErrors[24] := #bInError24;
   #abErrors[25] := #bInError25;
   #abErrors[26] := #bInError26;
   #abErrors[27] := #bInError27;
   #abErrors[28] := #bInError28;
   #abErrors[29] := #bInError29;
   #abErrors[30] := #bInError30;
   #bErrorExists := #bInError01 OR #bInError02 OR #bInError03 OR #bInError04 OR #bInError05 OR #bInError06 OR #bInError07 OR #bInError08 OR #bInError09 OR #bInError10 OR #bInError11 OR #bInError12 OR #bInError13 OR #bInError14 OR #bInError15 OR #bInError16 OR #bInError17 OR #bInError18 OR #bInError19 OR #bInError20 OR #bInError21 OR #bInError22 OR #bInError23 OR #bInError24 OR #bInError25 OR #bInError26 OR #bInError27 OR #bInError28 OR #bInError29 OR #bInError30;
END_REGION

REGION Network 3: Timer to change displayed error
   // ============================ Scroll errors on HMI ========================
   // Timed delay
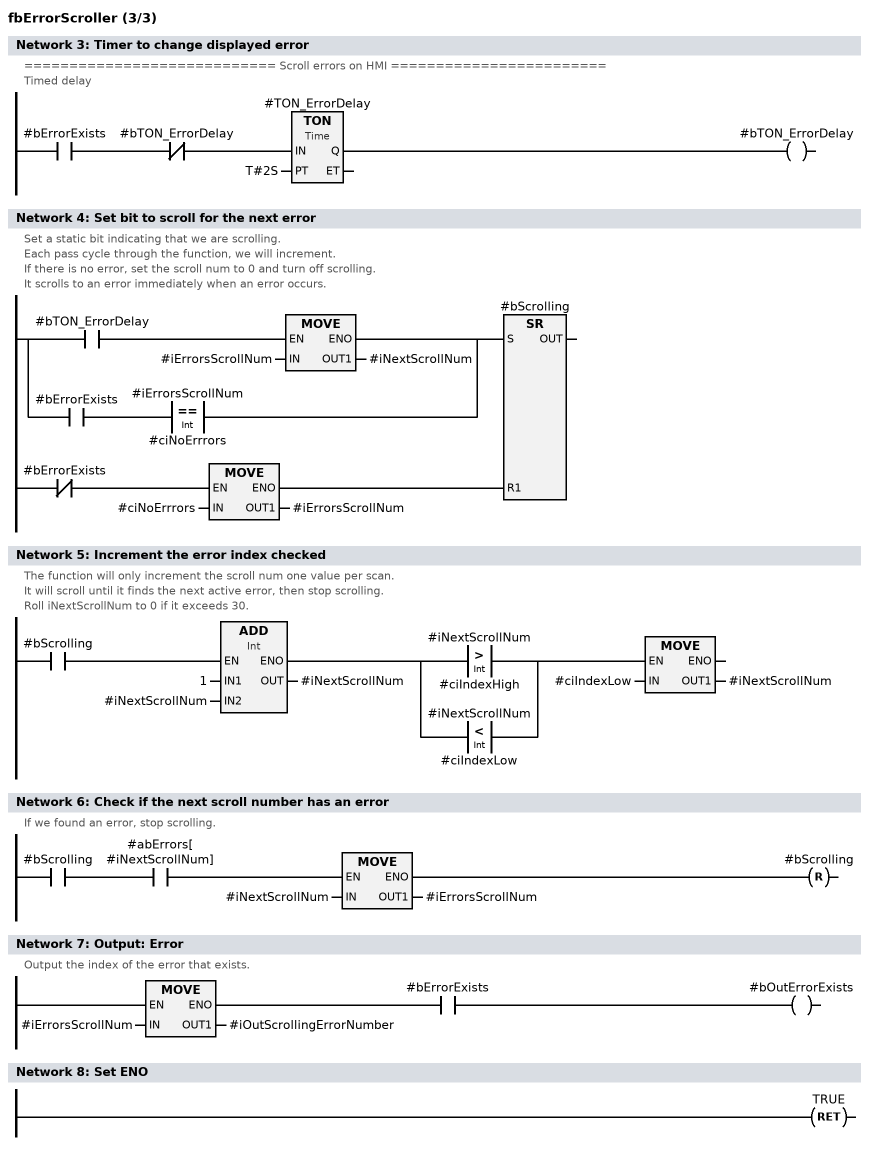
   RUNG wire#powerrail
      Contact( #bErrorExists )
      I_Contact( #bTON_ErrorDelay )
      { S7_Templates := "time_type := Time" } #TON_ErrorDelay.TON(pt := T#2S, et =>)
      Coil( #bTON_ErrorDelay )
   END_RUNG
   // the same network as SCL:
   #TON_ErrorDelay(IN := #bErrorExists AND NOT #bTON_ErrorDelay, PT := T#2S);   // TON
   #bTON_ErrorDelay := #TON_ErrorDelay.Q;
END_REGION

REGION Network 4: Set bit to scroll for the next error
   // Set a static bit indicating that we are scrolling.  
   // Each pass cycle through the function, we will increment.  
   // If there is no error, set the scroll num to 0 and turn off scrolling.  
   // It scrolls to an error immediately when an error occurs.
   RUNG wire#powerrail
      Contact( #bTON_ErrorDelay )
      { S7_GenerateENO := "TRUE" } Move(in := #iErrorsScrollNum, out1 => #iNextScrollNum)
      wire#w1
      S_SR(operand := #bScrolling, r1 := wire#w2)
   END_RUNG
   RUNG wire#powerrail
      Contact( #bErrorExists )
      { S7_Templates := "SrcType := Int" } EQ_Contact(in1 := #iErrorsScrollNum, in2 := #ciNoErrrors)
   END_RUNG wire#w1
   RUNG wire#powerrail
      I_Contact( #bErrorExists )
      { S7_GenerateENO := "TRUE" } Move(in := #ciNoErrrors, out1 => #iErrorsScrollNum)
   END_RUNG wire#w2
   // the same network as SCL:
   // ENO of a box is taken as its EN; it also drops when the box reports an error
   IF #bTON_ErrorDelay THEN #iNextScrollNum := #iErrorsScrollNum; END_IF;
   #_w1 := #bTON_ErrorDelay OR (#bErrorExists AND (#iErrorsScrollNum = #ciNoErrrors));
   IF NOT #bErrorExists THEN #iErrorsScrollNum := #ciNoErrrors; END_IF;
   IF #_w1 THEN
       #bScrolling := TRUE;   // SR flip-flop
   END_IF;
   IF NOT #bErrorExists THEN #bScrolling := FALSE; END_IF;
END_REGION

REGION Network 5: Increment the error index checked
   // The function will only increment the scroll num one value per scan.  
   // It will scroll until it finds the next active error, then stop scrolling.  
   // Roll iNextScrollNum to 0 if it exceeds 30.
   RUNG wire#powerrail
      Contact( #bScrolling )
      { S7_Templates := "SrcType := Int"; S7_GenerateENO := "TRUE" } Add(in1 := 1, in2 := #iNextScrollNum, out => #iNextScrollNum)
      wire#w1
      { S7_Templates := "SrcType := Int" } GT_Contact(in1 := #iNextScrollNum, in2 := #ciIndexHigh)
      wire#w2
      { S7_GenerateENO := "TRUE" } Move(in := #ciIndexLow, out1 => #iNextScrollNum)
   END_RUNG
   RUNG wire#w1
      { S7_Templates := "SrcType := Int" } LT_Contact(in1 := #iNextScrollNum, in2 := #ciIndexLow)
   END_RUNG wire#w2
   // the same network as SCL:
   // ENO of a box is taken as its EN; it also drops when the box reports an error
   IF #bScrolling THEN #iNextScrollNum := 1 + #iNextScrollNum; END_IF;
   IF #bScrolling AND ((#iNextScrollNum > #ciIndexHigh) OR (#iNextScrollNum < #ciIndexLow)) THEN
       #iNextScrollNum := #ciIndexLow;
   END_IF;
END_REGION

REGION Network 6: Check if the next scroll number has an error
   // If we found an error, stop scrolling.
   RUNG wire#powerrail
      Contact( #bScrolling )
      Contact( #abErrors[#iNextScrollNum] )
      { S7_GenerateENO := "TRUE" } Move(in := #iNextScrollNum, out1 => #iErrorsScrollNum)
      R_Coil( #bScrolling )
   END_RUNG
   // the same network as SCL:
   // ENO of a box is taken as its EN; it also drops when the box reports an error
   IF #bScrolling AND #abErrors[#iNextScrollNum] THEN
       #iErrorsScrollNum := #iNextScrollNum;
       #bScrolling := FALSE;
   END_IF;
END_REGION

REGION Network 7: Output: Error
   // Output the index of the error that exists.
   RUNG wire#powerrail
      { S7_GenerateENO := "TRUE" } Move(in := #iErrorsScrollNum, out1 => #iOutScrollingErrorNumber)
      Contact( #bErrorExists )
      Coil( #bOutErrorExists )
   END_RUNG
   // the same network as SCL:
   // ENO of a box is taken as its EN; it also drops when the box reports an error
   #iOutScrollingErrorNumber := #iErrorsScrollNum;
   #bOutErrorExists := #bErrorExists;
END_REGION

REGION Network 8: Set ENO
   RUNG wire#powerrail
      ReturnCoil( TRUE )
   END_RUNG
   // the same network as SCL:
   ENO := TRUE;
   RETURN;
END_REGION
END_FUNCTION_BLOCK

FUNCTION "fcSetHMIStatusSimulation" : Void   // FC333, LAD
TITLE = Sets HMI Status
{ S7_Optimized_Access := 'TRUE' }
VERSION : 0.1
// Wrapper function for setting the HMI status of a device
// 
// In order of priority:
// 1. E-stop
// 2. Error
// 3. Forward/Work Position
// 4. Reverse/Home Position
// 5. Forward/Work On
// 6. Reverse/Home On
// 7. None
// stored: AutoNumber true, IsIECCheckEnabled false, SetENOAutomatically false, UDAEnableTagReadback false
   VAR_INPUT
      bInEstop : Bool;
      bInError : Bool;
      bInForwardWork : Bool;
      bInReverseHome : Bool;
      bInOnForwardWork : Bool;
      bInOnReverseHome : Bool;
      bInSimulate : Bool;
   END_VAR
   VAR_OUTPUT
      iOutStatus : Int;
   END_VAR
BEGIN

REGION Network 1: Set Reverse/Home On
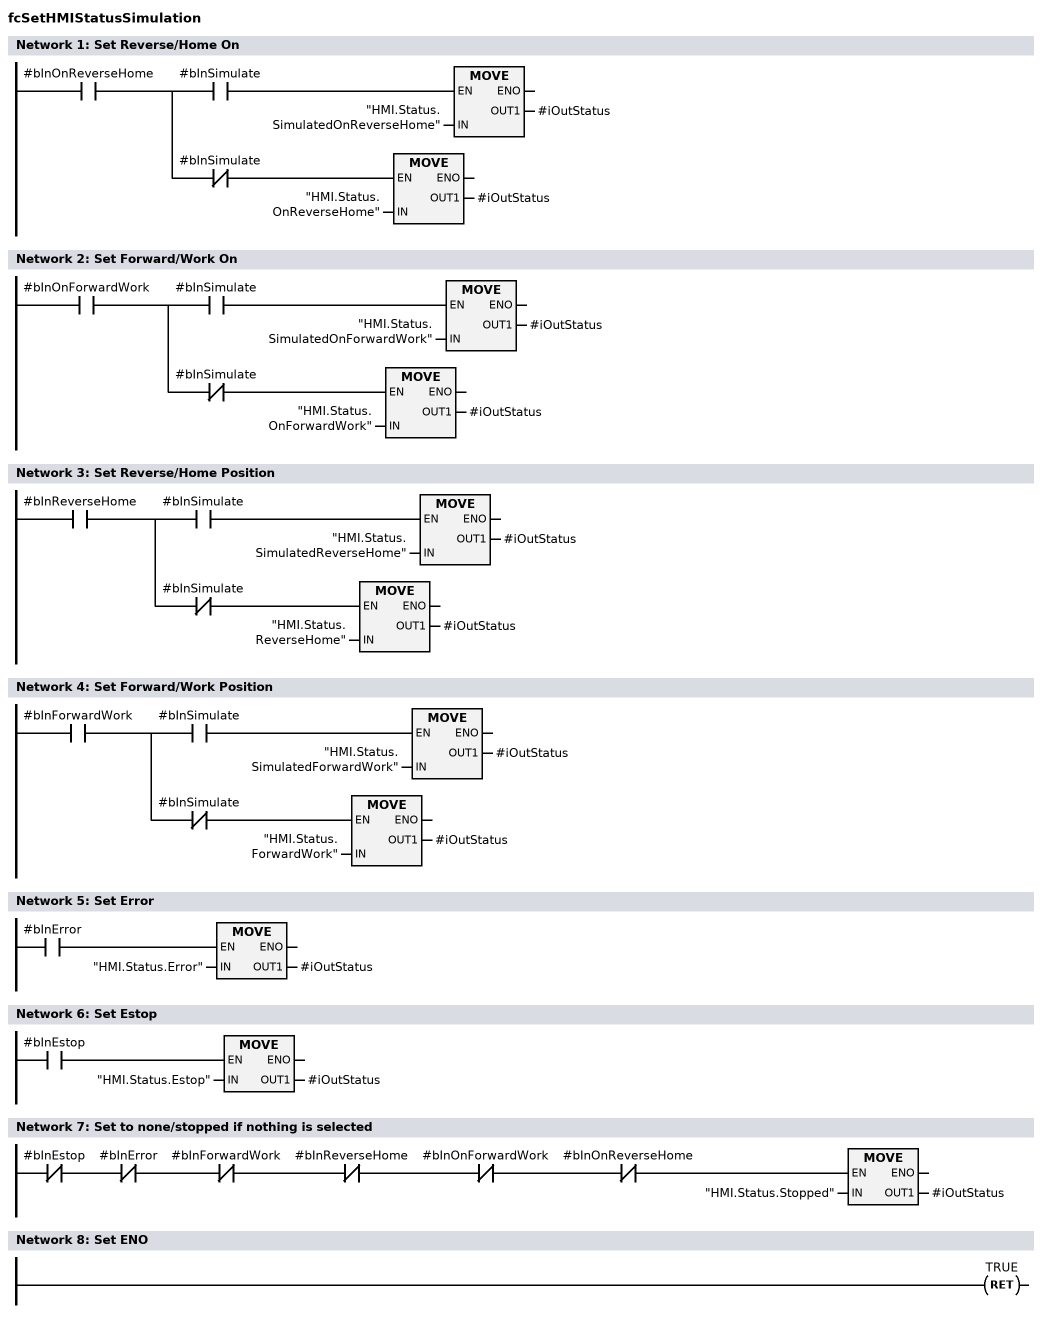
   RUNG wire#powerrail
      Contact( #bInOnReverseHome )
      wire#w1
      Contact( #bInSimulate )
      Move(in := "HMI.Status.SimulatedOnReverseHome", out1 => #iOutStatus)
   END_RUNG
   RUNG wire#w1
      I_Contact( #bInSimulate )
      Move(in := "HMI.Status.OnReverseHome", out1 => #iOutStatus)
   END_RUNG
   // the same network as SCL:
   IF #bInOnReverseHome AND #bInSimulate THEN #iOutStatus := "HMI.Status.SimulatedOnReverseHome"; END_IF;
   IF #bInOnReverseHome AND NOT #bInSimulate THEN #iOutStatus := "HMI.Status.OnReverseHome"; END_IF;
END_REGION

REGION Network 2: Set Forward/Work On
   RUNG wire#powerrail
      Contact( #bInOnForwardWork )
      wire#w1
      Contact( #bInSimulate )
      Move(in := "HMI.Status.SimulatedOnForwardWork", out1 => #iOutStatus)
   END_RUNG
   RUNG wire#w1
      I_Contact( #bInSimulate )
      Move(in := "HMI.Status.OnForwardWork", out1 => #iOutStatus)
   END_RUNG
   // the same network as SCL:
   IF #bInOnForwardWork AND #bInSimulate THEN #iOutStatus := "HMI.Status.SimulatedOnForwardWork"; END_IF;
   IF #bInOnForwardWork AND NOT #bInSimulate THEN #iOutStatus := "HMI.Status.OnForwardWork"; END_IF;
END_REGION

REGION Network 3: Set Reverse/Home Position
   RUNG wire#powerrail
      Contact( #bInReverseHome )
      wire#w1
      Contact( #bInSimulate )
      Move(in := "HMI.Status.SimulatedReverseHome", out1 => #iOutStatus)
   END_RUNG
   RUNG wire#w1
      I_Contact( #bInSimulate )
      Move(in := "HMI.Status.ReverseHome", out1 => #iOutStatus)
   END_RUNG
   // the same network as SCL:
   IF #bInReverseHome AND #bInSimulate THEN #iOutStatus := "HMI.Status.SimulatedReverseHome"; END_IF;
   IF #bInReverseHome AND NOT #bInSimulate THEN #iOutStatus := "HMI.Status.ReverseHome"; END_IF;
END_REGION

REGION Network 4: Set Forward/Work Position
   RUNG wire#powerrail
      Contact( #bInForwardWork )
      wire#w1
      Contact( #bInSimulate )
      Move(in := "HMI.Status.SimulatedForwardWork", out1 => #iOutStatus)
   END_RUNG
   RUNG wire#w1
      I_Contact( #bInSimulate )
      Move(in := "HMI.Status.ForwardWork", out1 => #iOutStatus)
   END_RUNG
   // the same network as SCL:
   IF #bInForwardWork AND #bInSimulate THEN #iOutStatus := "HMI.Status.SimulatedForwardWork"; END_IF;
   IF #bInForwardWork AND NOT #bInSimulate THEN #iOutStatus := "HMI.Status.ForwardWork"; END_IF;
END_REGION

REGION Network 5: Set Error
   RUNG wire#powerrail
      Contact( #bInError )
      Move(in := "HMI.Status.Error", out1 => #iOutStatus)
   END_RUNG
   // the same network as SCL:
   IF #bInError THEN #iOutStatus := "HMI.Status.Error"; END_IF;
END_REGION

REGION Network 6: Set Estop
   RUNG wire#powerrail
      Contact( #bInEstop )
      Move(in := "HMI.Status.Estop", out1 => #iOutStatus)
   END_RUNG
   // the same network as SCL:
   IF #bInEstop THEN #iOutStatus := "HMI.Status.Estop"; END_IF;
END_REGION

REGION Network 7: Set to none/stopped if nothing is selected
   RUNG wire#powerrail
      I_Contact( #bInEstop )
      I_Contact( #bInError )
      I_Contact( #bInForwardWork )
      I_Contact( #bInReverseHome )
      I_Contact( #bInOnForwardWork )
      I_Contact( #bInOnReverseHome )
      Move(in := "HMI.Status.Stopped", out1 => #iOutStatus)
   END_RUNG
   // the same network as SCL:
   IF NOT #bInEstop AND NOT #bInError AND NOT #bInForwardWork AND NOT #bInReverseHome AND NOT #bInOnForwardWork AND NOT #bInOnReverseHome THEN
       #iOutStatus := "HMI.Status.Stopped";
   END_IF;
END_REGION

REGION Network 8: Set ENO
   RUNG wire#powerrail
      ReturnCoil( TRUE )
   END_RUNG
   // the same network as SCL:
   ENO := TRUE;
   RETURN;
END_REGION
END_FUNCTION

FUNCTION "fcBitsToWord" : Void   // FC301, LAD
TITLE = Pack Bits into word
{ S7_Optimized_Access := 'TRUE' }
AUTHOR : DMC
FAMILY : LowLevel
VERSION : 0.1
// stored: AutoNumber false, IsIECCheckEnabled false, SetENOAutomatically false, UDAEnableTagReadback false
   VAR_INPUT
      bInBit00 : Bool;   // Bit 0
      bInBit01 : Bool;   // Bit 1
      bInBit02 : Bool;   // Bit 2
      bInBit03 : Bool;   // Bit 3
      bInBit04 : Bool;   // Bit 4
      bInBit05 : Bool;   // Bit 5
      bInBit06 : Bool;   // Bit 6
      bInBit07 : Bool;   // Bit 7
      bInBit08 : Bool;   // Bit 8
      bInBit09 : Bool;   // Bit 9
      bInBit10 : Bool;   // Bit 10
      bInBit11 : Bool;   // Bit 11
      bInBit12 : Bool;   // Bit 12
      bInBit13 : Bool;   // Bit 13
      bInBit14 : Bool;   // Bit 14
      bInBit15 : Bool;   // Bit 15
   END_VAR
   VAR_OUTPUT
      wOutWord : Word;   // Packed Word
   END_VAR
BEGIN

REGION Network 1: Bit0
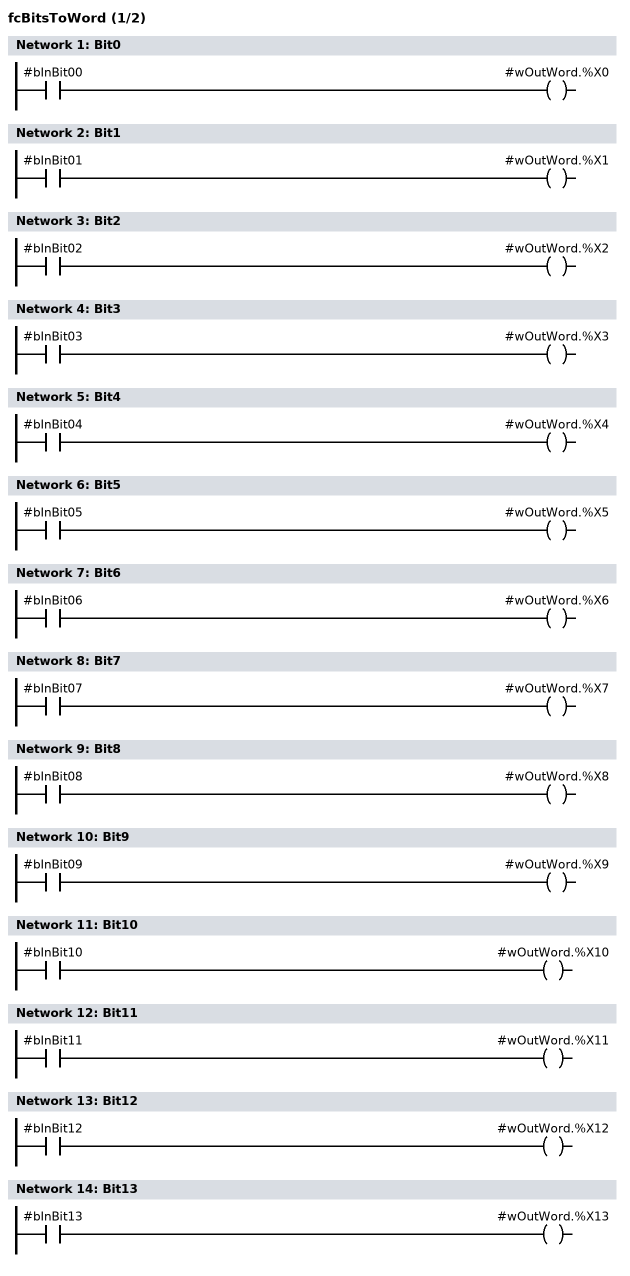
   RUNG wire#powerrail
      Contact( #bInBit00 )
      Coil( #wOutWord.%X0 )
   END_RUNG
   // the same network as SCL:
   #wOutWord.%X0 := #bInBit00;
END_REGION

REGION Network 2: Bit1
   RUNG wire#powerrail
      Contact( #bInBit01 )
      Coil( #wOutWord.%X1 )
   END_RUNG
   // the same network as SCL:
   #wOutWord.%X1 := #bInBit01;
END_REGION

REGION Network 3: Bit2
   RUNG wire#powerrail
      Contact( #bInBit02 )
      Coil( #wOutWord.%X2 )
   END_RUNG
   // the same network as SCL:
   #wOutWord.%X2 := #bInBit02;
END_REGION

REGION Network 4: Bit3
   RUNG wire#powerrail
      Contact( #bInBit03 )
      Coil( #wOutWord.%X3 )
   END_RUNG
   // the same network as SCL:
   #wOutWord.%X3 := #bInBit03;
END_REGION

REGION Network 5: Bit4
   RUNG wire#powerrail
      Contact( #bInBit04 )
      Coil( #wOutWord.%X4 )
   END_RUNG
   // the same network as SCL:
   #wOutWord.%X4 := #bInBit04;
END_REGION

REGION Network 6: Bit5
   RUNG wire#powerrail
      Contact( #bInBit05 )
      Coil( #wOutWord.%X5 )
   END_RUNG
   // the same network as SCL:
   #wOutWord.%X5 := #bInBit05;
END_REGION

REGION Network 7: Bit6
   RUNG wire#powerrail
      Contact( #bInBit06 )
      Coil( #wOutWord.%X6 )
   END_RUNG
   // the same network as SCL:
   #wOutWord.%X6 := #bInBit06;
END_REGION

REGION Network 8: Bit7
   RUNG wire#powerrail
      Contact( #bInBit07 )
      Coil( #wOutWord.%X7 )
   END_RUNG
   // the same network as SCL:
   #wOutWord.%X7 := #bInBit07;
END_REGION

REGION Network 9: Bit8
   RUNG wire#powerrail
      Contact( #bInBit08 )
      Coil( #wOutWord.%X8 )
   END_RUNG
   // the same network as SCL:
   #wOutWord.%X8 := #bInBit08;
END_REGION

REGION Network 10: Bit9
   RUNG wire#powerrail
      Contact( #bInBit09 )
      Coil( #wOutWord.%X9 )
   END_RUNG
   // the same network as SCL:
   #wOutWord.%X9 := #bInBit09;
END_REGION

REGION Network 11: Bit10
   RUNG wire#powerrail
      Contact( #bInBit10 )
      Coil( #wOutWord.%X10 )
   END_RUNG
   // the same network as SCL:
   #wOutWord.%X10 := #bInBit10;
END_REGION

REGION Network 12: Bit11
   RUNG wire#powerrail
      Contact( #bInBit11 )
      Coil( #wOutWord.%X11 )
   END_RUNG
   // the same network as SCL:
   #wOutWord.%X11 := #bInBit11;
END_REGION

REGION Network 13: Bit12
   RUNG wire#powerrail
      Contact( #bInBit12 )
      Coil( #wOutWord.%X12 )
   END_RUNG
   // the same network as SCL:
   #wOutWord.%X12 := #bInBit12;
END_REGION

REGION Network 14: Bit13
   RUNG wire#powerrail
      Contact( #bInBit13 )
      Coil( #wOutWord.%X13 )
   END_RUNG
   // the same network as SCL:
   #wOutWord.%X13 := #bInBit13;
END_REGION

REGION Network 15: Bit14
